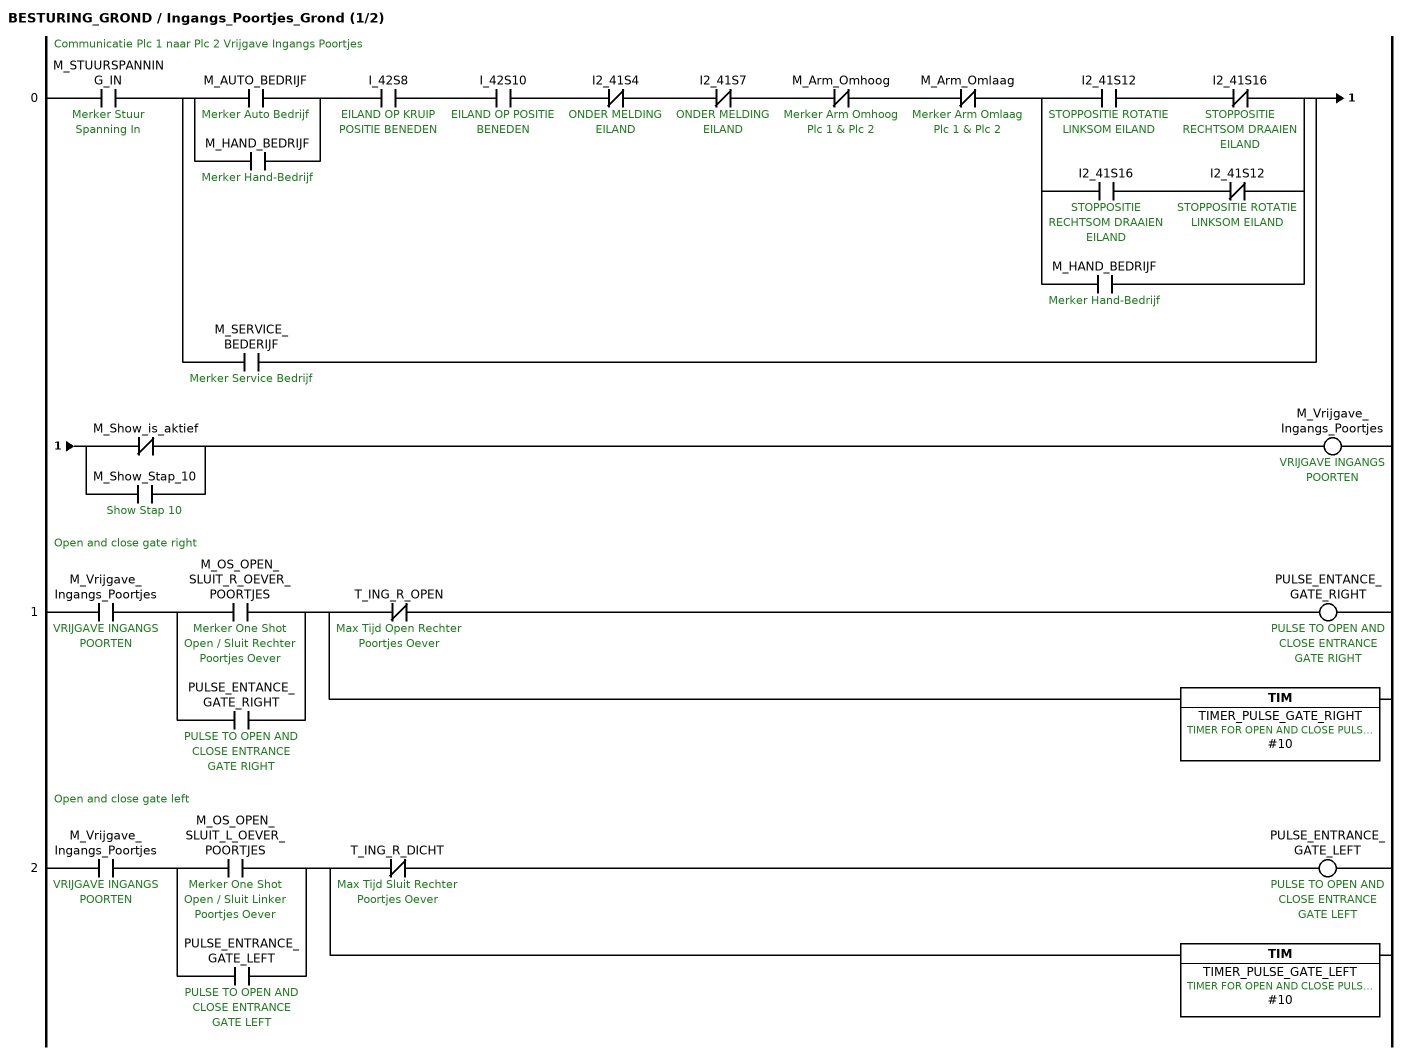
; [picture p349: BESTURING_GROND / Ingangs_Poortjes_Grond, rungs 0-2]
; rung 0: Communicatie Plc 1 naar Plc 2 Vrijgave Ingangs Poortjes
LD M_STUURSPANNING_IN  ; Merker Stuur Spanning In
LD M_AUTO_BEDRIJF  ; Merker Auto Bedrijf
OR M_HAND_BEDRIJF  ; Merker Hand-Bedrijf
AND I_42S8  ; EILAND OP KRUIP POSITIE BENEDEN
AND I_42S10  ; EILAND OP POSITIE BENEDEN
ANDNOT I2_41S4  ; ONDER MELDING EILAND
ANDNOT I2_41S7  ; ONDER MELDING EILAND
ANDNOT M_Arm_Omhoog  ; Merker Arm Omhoog Plc 1 & Plc 2
ANDNOT M_Arm_Omlaag  ; Merker Arm Omlaag Plc 1 & Plc 2
LD I2_41S12  ; STOPPOSITIE ROTATIE LINKSOM EILAND
ANDNOT I2_41S16  ; STOPPOSITIE RECHTSOM DRAAIEN EILAND
LD I2_41S16  ; STOPPOSITIE RECHTSOM DRAAIEN EILAND
ANDNOT I2_41S12  ; STOPPOSITIE ROTATIE LINKSOM EILAND
ORLD
OR M_HAND_BEDRIJF  ; Merker Hand-Bedrijf
ANDLD
OR M_SERVICE_BEDERIJF  ; Merker Service Bedrijf
ANDLD
LDNOT M_Show_is_aktief
OR M_Show_Stap_10  ; Show Stap 10
ANDLD
OUT M_Vrijgave_Ingangs_Poortjes  ; VRIJGAVE INGANGS POORTEN
; rung 1: Open and close gate right
LD M_Vrijgave_Ingangs_Poortjes  ; VRIJGAVE INGANGS POORTEN
LD M_OS_OPEN_SLUIT_R_OEVER_POORTJES  ; Merker One Shot Open / Sluit Rechter Poortjes Oever
OR PULSE_ENTANCE_GATE_RIGHT  ; PULSE TO OPEN AND CLOSE ENTRANCE GATE RIGHT
ANDLD
OUT TR0
ANDNOT T_ING_R_OPEN  ; Max Tijd Open Rechter Poortjes Oever
OUT PULSE_ENTANCE_GATE_RIGHT  ; PULSE TO OPEN AND CLOSE ENTRANCE GATE RIGHT
LD TR0
TIM TIMER_PULSE_GATE_RIGHT #10  ; TIMER FOR OPEN AND CLOSE PULSE ENTRANCE GATE RIGHT
; rung 2: Open and close gate left
LD M_Vrijgave_Ingangs_Poortjes  ; VRIJGAVE INGANGS POORTEN
LD M_OS_OPEN_SLUIT_L_OEVER_POORTJES  ; Merker One Shot Open / Sluit Linker Poortjes Oever
OR PULSE_ENTRANCE_GATE_LEFT  ; PULSE TO OPEN AND CLOSE ENTRANCE GATE LEFT
ANDLD
OUT TR0
ANDNOT T_ING_R_DICHT  ; Max Tijd Sluit Rechter Poortjes Oever
OUT PULSE_ENTRANCE_GATE_LEFT  ; PULSE TO OPEN AND CLOSE ENTRANCE GATE LEFT
LD TR0
TIM TIMER_PULSE_GATE_LEFT #10  ; TIMER FOR OPEN AND CLOSE PULSE ENTRANCE GATE LEFT

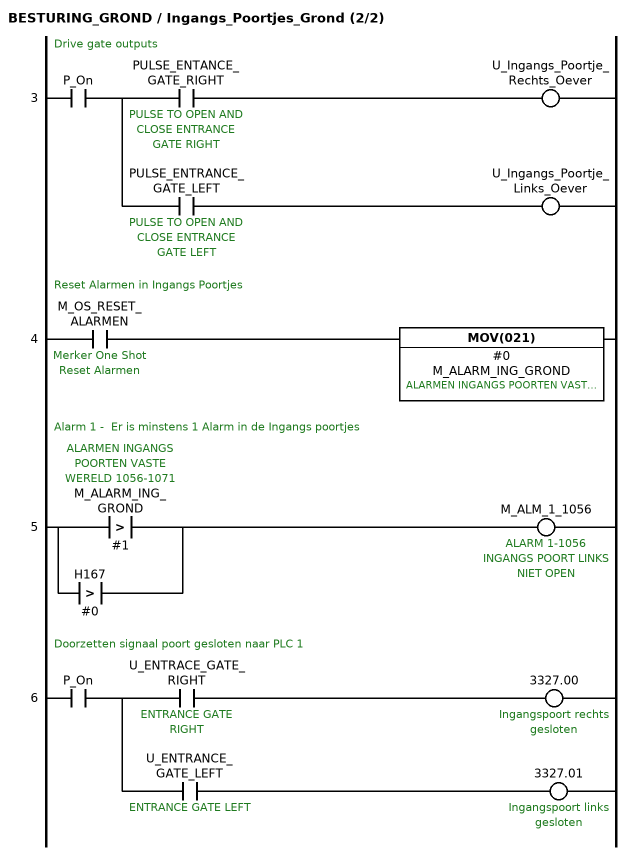
; rung 3: Drive gate outputs
LD P_On
OUT TR0
AND PULSE_ENTANCE_GATE_RIGHT  ; PULSE TO OPEN AND CLOSE ENTRANCE GATE RIGHT
OUT U_Ingangs_Poortje_Rechts_Oever
LD TR0
AND PULSE_ENTRANCE_GATE_LEFT  ; PULSE TO OPEN AND CLOSE ENTRANCE GATE LEFT
OUT U_Ingangs_Poortje_Links_Oever
; rung 4: Reset Alarmen in Ingangs Poortjes
LD M_OS_RESET_ALARMEN  ; Merker One Shot Reset Alarmen
MOV(021) #0 M_ALARM_ING_GROND  ; ALARMEN INGANGS POORTEN VASTE WERELD 1056-1071
; rung 5: Alarm 1 -  Er is minstens 1 Alarm in de Ingangs poortjes
LD>(320) M_ALARM_ING_GROND #1  ; ALARMEN INGANGS POORTEN VASTE WERELD 1056-1071
OR>(320) H167 #0
OUT M_ALM_1_1056  ; ALARM 1-1056 INGANGS POORT LINKS NIET OPEN
; rung 6: Doorzetten signaal poort gesloten naar PLC 1
LD P_On
OUT TR0
AND U_ENTRACE_GATE_RIGHT  ; ENTRANCE GATE RIGHT
OUT 3327.00  ; Ingangspoort rechts gesloten
LD TR0
AND U_ENTRANCE_GATE_LEFT  ; ENTRANCE GATE LEFT
OUT 3327.01  ; Ingangspoort links gesloten

### Section Uitgangs_poortjes_Grond

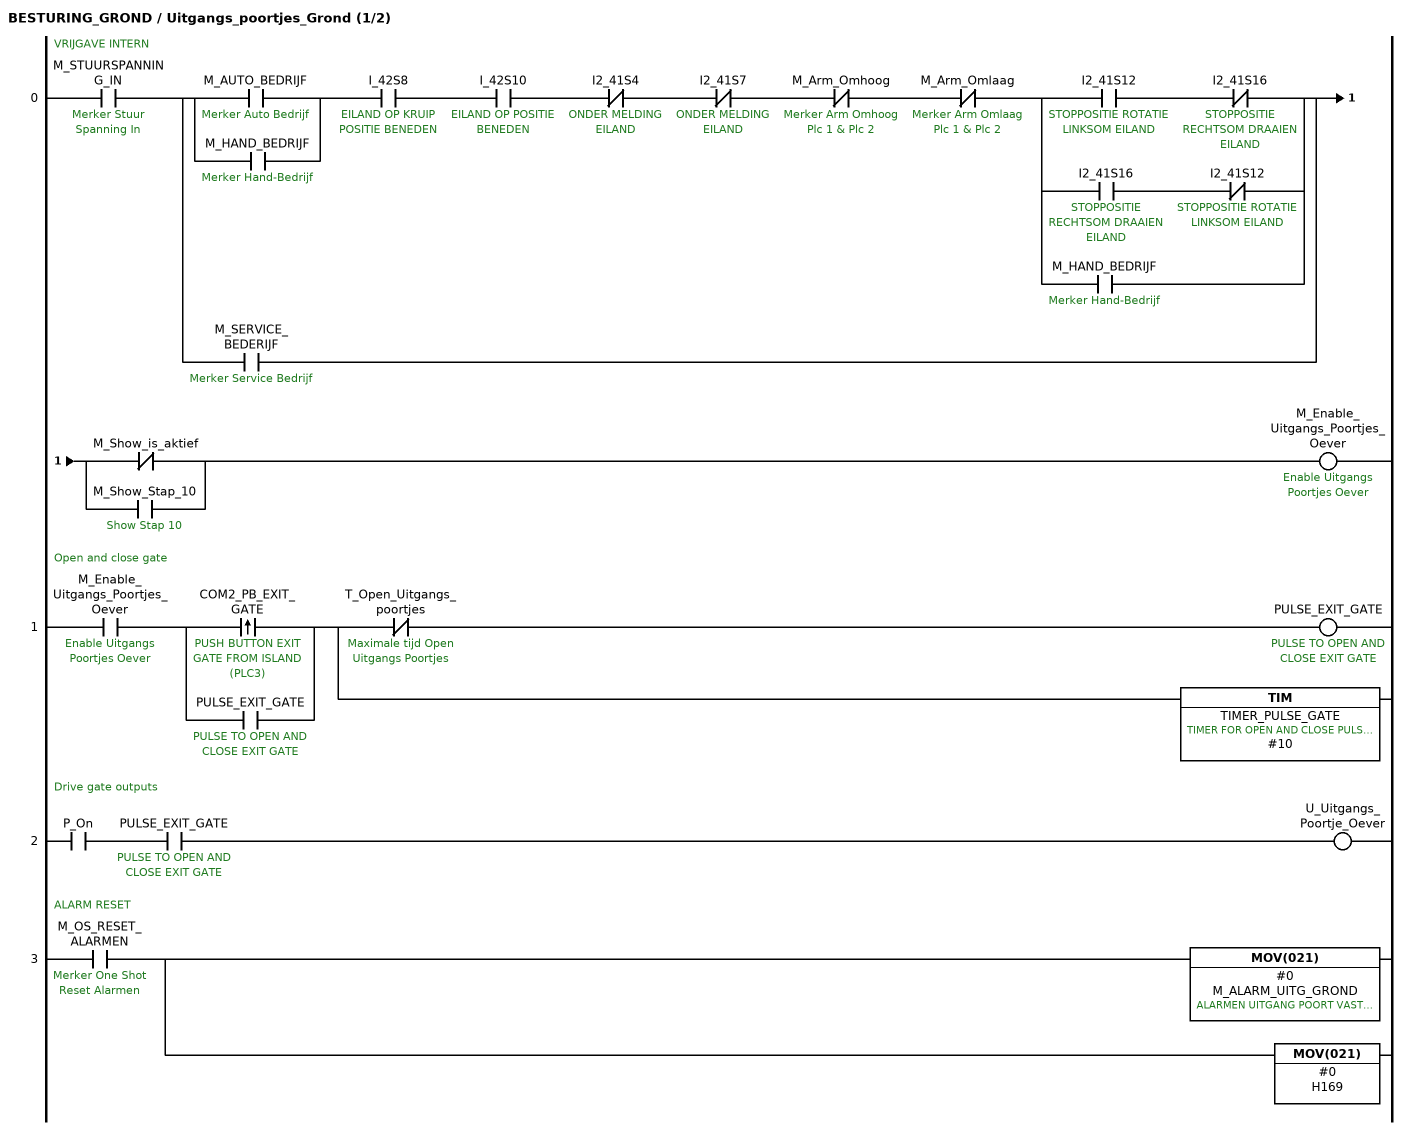
; rung 0: VRIJGAVE INTERN
LD M_STUURSPANNING_IN  ; Merker Stuur Spanning In
LD M_AUTO_BEDRIJF  ; Merker Auto Bedrijf
OR M_HAND_BEDRIJF  ; Merker Hand-Bedrijf
AND I_42S8  ; EILAND OP KRUIP POSITIE BENEDEN
AND I_42S10  ; EILAND OP POSITIE BENEDEN
ANDNOT I2_41S4  ; ONDER MELDING EILAND
ANDNOT I2_41S7  ; ONDER MELDING EILAND
ANDNOT M_Arm_Omhoog  ; Merker Arm Omhoog Plc 1 & Plc 2
ANDNOT M_Arm_Omlaag  ; Merker Arm Omlaag Plc 1 & Plc 2
LD I2_41S12  ; STOPPOSITIE ROTATIE LINKSOM EILAND
ANDNOT I2_41S16  ; STOPPOSITIE RECHTSOM DRAAIEN EILAND
LD I2_41S16  ; STOPPOSITIE RECHTSOM DRAAIEN EILAND
ANDNOT I2_41S12  ; STOPPOSITIE ROTATIE LINKSOM EILAND
ORLD
OR M_HAND_BEDRIJF  ; Merker Hand-Bedrijf
ANDLD
OR M_SERVICE_BEDERIJF  ; Merker Service Bedrijf
ANDLD
LDNOT M_Show_is_aktief
OR M_Show_Stap_10  ; Show Stap 10
ANDLD
OUT M_Enable_Uitgangs_Poortjes_Oever  ; Enable Uitgangs Poortjes Oever
; rung 1: Open and close gate
LD M_Enable_Uitgangs_Poortjes_Oever  ; Enable Uitgangs Poortjes Oever
@LD COM2_PB_EXIT_GATE  ; PUSH BUTTON EXIT GATE FROM ISLAND (PLC3)
OR PULSE_EXIT_GATE  ; PULSE TO OPEN AND CLOSE EXIT GATE
ANDLD
OUT TR0
ANDNOT T_Open_Uitgangs_poortjes  ; Maximale tijd Open Uitgangs Poortjes
OUT PULSE_EXIT_GATE  ; PULSE TO OPEN AND CLOSE EXIT GATE
LD TR0
TIM TIMER_PULSE_GATE #10  ; TIMER FOR OPEN AND CLOSE PULSE EXIT GATE
; rung 2: Drive gate outputs
LD P_On
AND PULSE_EXIT_GATE  ; PULSE TO OPEN AND CLOSE EXIT GATE
OUT U_Uitgangs_Poortje_Oever
; rung 3: ALARM RESET
LD M_OS_RESET_ALARMEN  ; Merker One Shot Reset Alarmen
MOV(021) #0 M_ALARM_UITG_GROND  ; ALARMEN UITGANG POORT VASTE WERELD 1088-1103
MOV(021) #0 H169

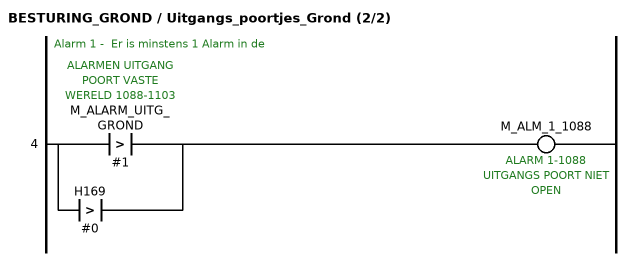
; rung 4: Alarm 1 -  Er is minstens 1 Alarm in de
LD>(320) M_ALARM_UITG_GROND #1  ; ALARMEN UITGANG POORT VASTE WERELD 1088-1103
OR>(320) H169 #0
OUT M_ALM_1_1088  ; ALARM 1-1088 UITGANGS POORT NIET OPEN

### Section Hydrauliek_Arm

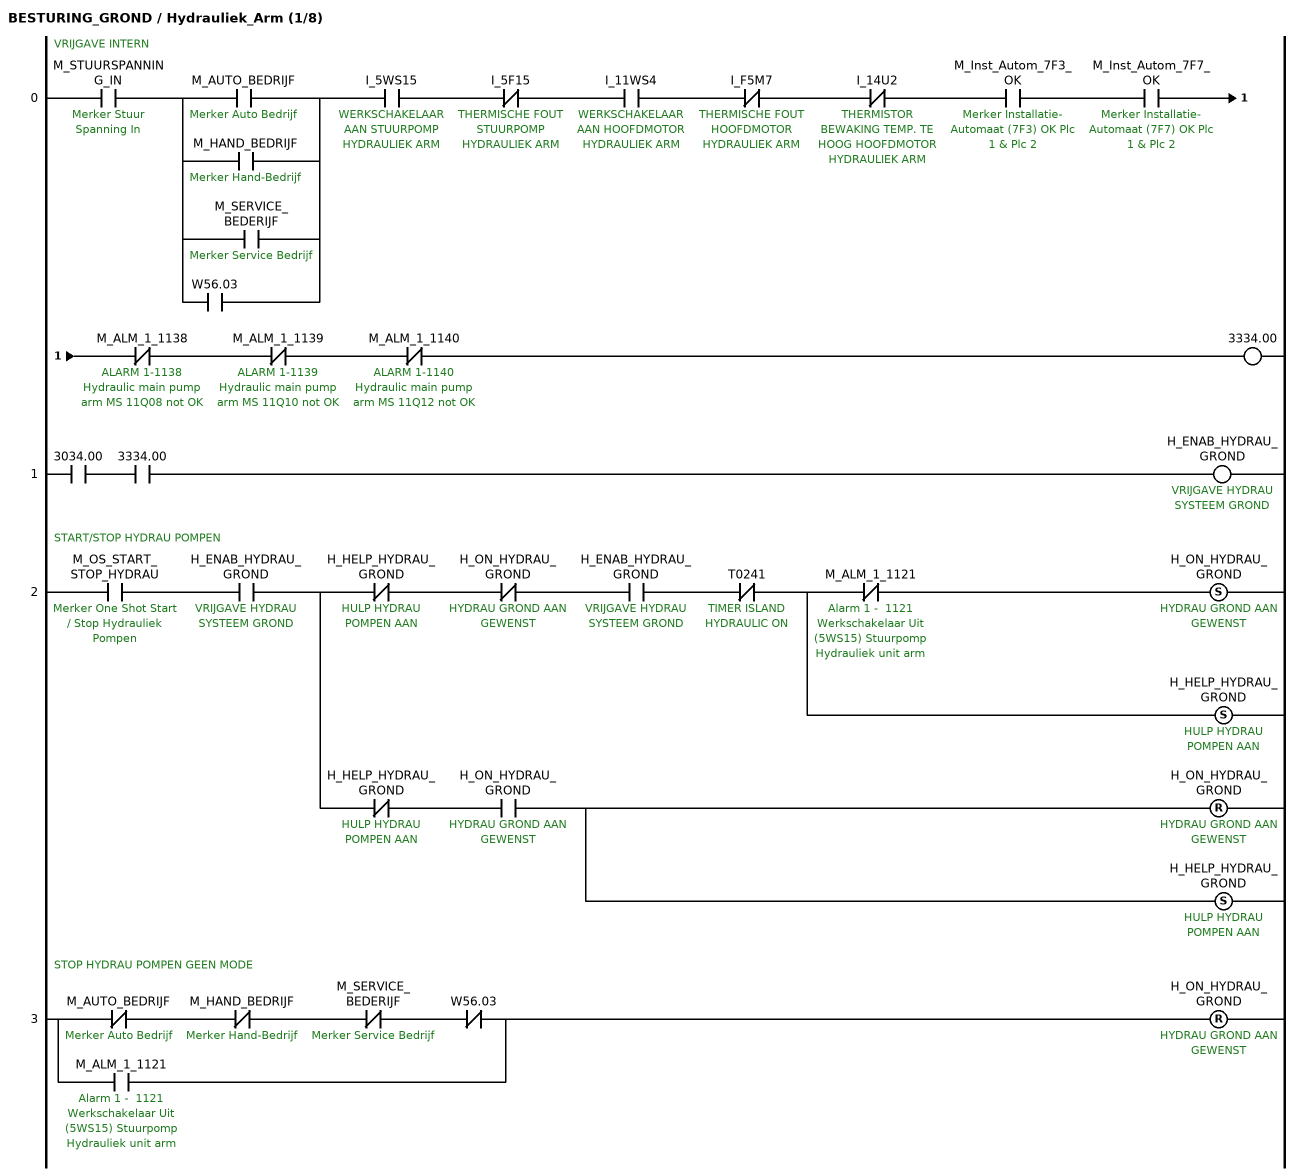
; rung 0: VRIJGAVE INTERN
LD M_STUURSPANNING_IN  ; Merker Stuur Spanning In
LD M_AUTO_BEDRIJF  ; Merker Auto Bedrijf
OR M_HAND_BEDRIJF  ; Merker Hand-Bedrijf
OR M_SERVICE_BEDERIJF  ; Merker Service Bedrijf
OR W56.03
ANDLD
AND I_5WS15  ; WERKSCHAKELAAR AAN STUURPOMP HYDRAULIEK ARM
ANDNOT I_5F15  ; THERMISCHE FOUT STUURPOMP HYDRAULIEK ARM
AND I_11WS4  ; WERKSCHAKELAAR AAN HOOFDMOTOR HYDRAULIEK ARM
ANDNOT I_F5M7  ; THERMISCHE FOUT HOOFDMOTOR HYDRAULIEK ARM
ANDNOT I_14U2  ; THERMISTOR BEWAKING TEMP. TE HOOG HOOFDMOTOR HYDRAULIEK ARM
AND M_Inst_Autom_7F3_OK  ; Merker Installatie-Automaat (7F3) OK Plc 1 & Plc 2
AND M_Inst_Autom_7F7_OK  ; Merker Installatie-Automaat (7F7) OK Plc 1 & Plc 2
ANDNOT M_ALM_1_1138  ; ALARM 1-1138 Hydraulic main pump arm MS 11Q08 not OK
ANDNOT M_ALM_1_1139  ; ALARM 1-1139 Hydraulic main pump arm MS 11Q10 not OK
ANDNOT M_ALM_1_1140  ; ALARM 1-1140 Hydraulic main pump arm MS 11Q12 not OK
OUT 3334.00
; rung 1
LD 3034.00
AND 3334.00
OUT H_ENAB_HYDRAU_GROND  ; VRIJGAVE HYDRAU SYSTEEM GROND
; rung 2: START/STOP HYDRAU POMPEN
LD M_OS_START_STOP_HYDRAU  ; Merker One Shot Start / Stop Hydrauliek Pompen
AND H_ENAB_HYDRAU_GROND  ; VRIJGAVE HYDRAU SYSTEEM GROND
OUT TR0
ANDNOT H_HELP_HYDRAU_GROND  ; HULP HYDRAU POMPEN AAN
ANDNOT H_ON_HYDRAU_GROND  ; HYDRAU GROND AAN GEWENST
AND H_ENAB_HYDRAU_GROND  ; VRIJGAVE HYDRAU SYSTEEM GROND
ANDNOT T0241  ; TIMER ISLAND HYDRAULIC ON
OUT TR1
ANDNOT M_ALM_1_1121  ; Alarm 1 -  1121 Werkschakelaar Uit (5WS15) Stuurpomp Hydrauliek unit arm
SET H_ON_HYDRAU_GROND  ; HYDRAU GROND AAN GEWENST
LD TR1
SET H_HELP_HYDRAU_GROND  ; HULP HYDRAU POMPEN AAN
LD TR0
ANDNOT H_HELP_HYDRAU_GROND  ; HULP HYDRAU POMPEN AAN
AND H_ON_HYDRAU_GROND  ; HYDRAU GROND AAN GEWENST
RSET H_ON_HYDRAU_GROND  ; HYDRAU GROND AAN GEWENST
SET H_HELP_HYDRAU_GROND  ; HULP HYDRAU POMPEN AAN
; rung 3: STOP HYDRAU POMPEN GEEN MODE
LDNOT M_AUTO_BEDRIJF  ; Merker Auto Bedrijf
ANDNOT M_HAND_BEDRIJF  ; Merker Hand-Bedrijf
ANDNOT M_SERVICE_BEDERIJF  ; Merker Service Bedrijf
ANDNOT W56.03
OR M_ALM_1_1121  ; Alarm 1 -  1121 Werkschakelaar Uit (5WS15) Stuurpomp Hydrauliek unit arm
RSET H_ON_HYDRAU_GROND  ; HYDRAU GROND AAN GEWENST

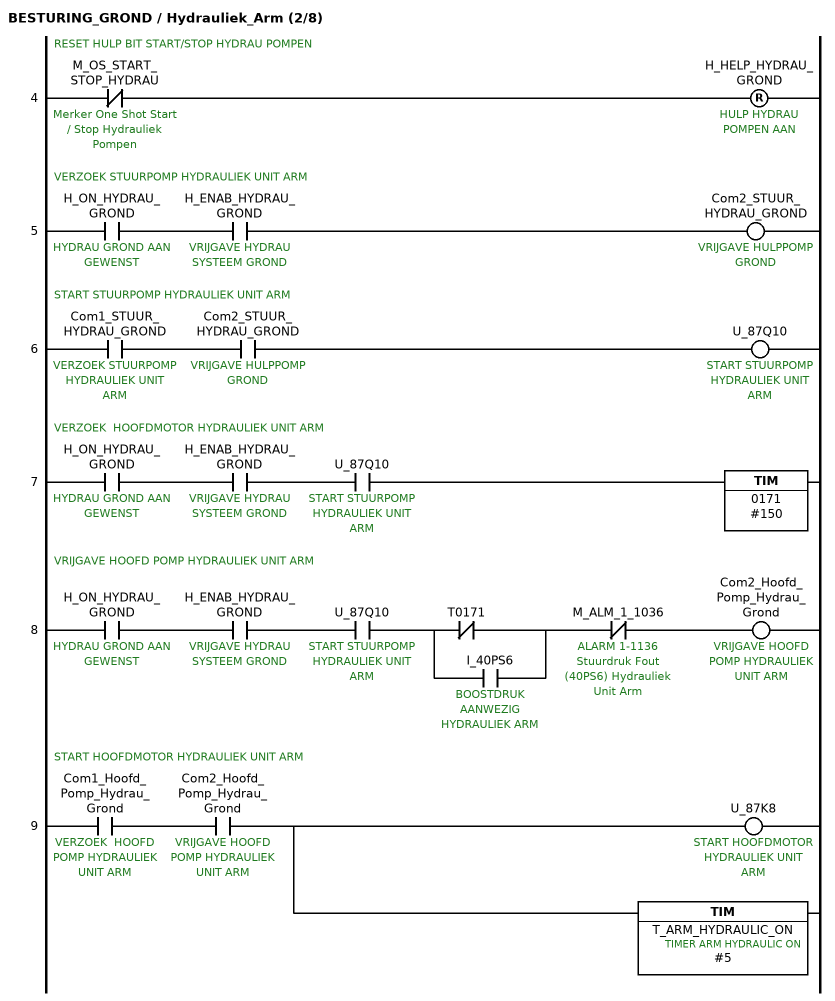
; rung 4: RESET HULP BIT START/STOP HYDRAU POMPEN
LDNOT M_OS_START_STOP_HYDRAU  ; Merker One Shot Start / Stop Hydrauliek Pompen
RSET H_HELP_HYDRAU_GROND  ; HULP HYDRAU POMPEN AAN
; rung 5: VERZOEK STUURPOMP HYDRAULIEK UNIT ARM
LD H_ON_HYDRAU_GROND  ; HYDRAU GROND AAN GEWENST
AND H_ENAB_HYDRAU_GROND  ; VRIJGAVE HYDRAU SYSTEEM GROND
OUT Com2_STUUR_HYDRAU_GROND  ; VRIJGAVE HULPPOMP GROND
; rung 6: START STUURPOMP HYDRAULIEK UNIT ARM
LD Com1_STUUR_HYDRAU_GROND  ; VERZOEK STUURPOMP HYDRAULIEK UNIT ARM
AND Com2_STUUR_HYDRAU_GROND  ; VRIJGAVE HULPPOMP GROND
OUT U_87Q10  ; START STUURPOMP HYDRAULIEK UNIT ARM
; rung 7: VERZOEK  HOOFDMOTOR HYDRAULIEK UNIT ARM
LD H_ON_HYDRAU_GROND  ; HYDRAU GROND AAN GEWENST
AND H_ENAB_HYDRAU_GROND  ; VRIJGAVE HYDRAU SYSTEEM GROND
AND U_87Q10  ; START STUURPOMP HYDRAULIEK UNIT ARM
TIM 0171 #150
; rung 8: VRIJGAVE HOOFD POMP HYDRAULIEK UNIT ARM
LD H_ON_HYDRAU_GROND  ; HYDRAU GROND AAN GEWENST
AND H_ENAB_HYDRAU_GROND  ; VRIJGAVE HYDRAU SYSTEEM GROND
AND U_87Q10  ; START STUURPOMP HYDRAULIEK UNIT ARM
LDNOT T0171
OR I_40PS6  ; BOOSTDRUK AANWEZIG HYDRAULIEK ARM
ANDLD
ANDNOT M_ALM_1_1036  ; ALARM 1-1136 Stuurdruk Fout (40PS6) Hydrauliek Unit Arm
OUT Com2_Hoofd_Pomp_Hydrau_Grond  ; VRIJGAVE HOOFD POMP HYDRAULIEK UNIT ARM
; rung 9: START HOOFDMOTOR HYDRAULIEK UNIT ARM
LD Com1_Hoofd_Pomp_Hydrau_Grond  ; VERZOEK  HOOFD POMP HYDRAULIEK UNIT ARM
AND Com2_Hoofd_Pomp_Hydrau_Grond  ; VRIJGAVE HOOFD POMP HYDRAULIEK UNIT ARM
OUT U_87K8  ; START HOOFDMOTOR HYDRAULIEK UNIT ARM
TIM T_ARM_HYDRAULIC_ON #5  ; TIMER ARM HYDRAULIC ON

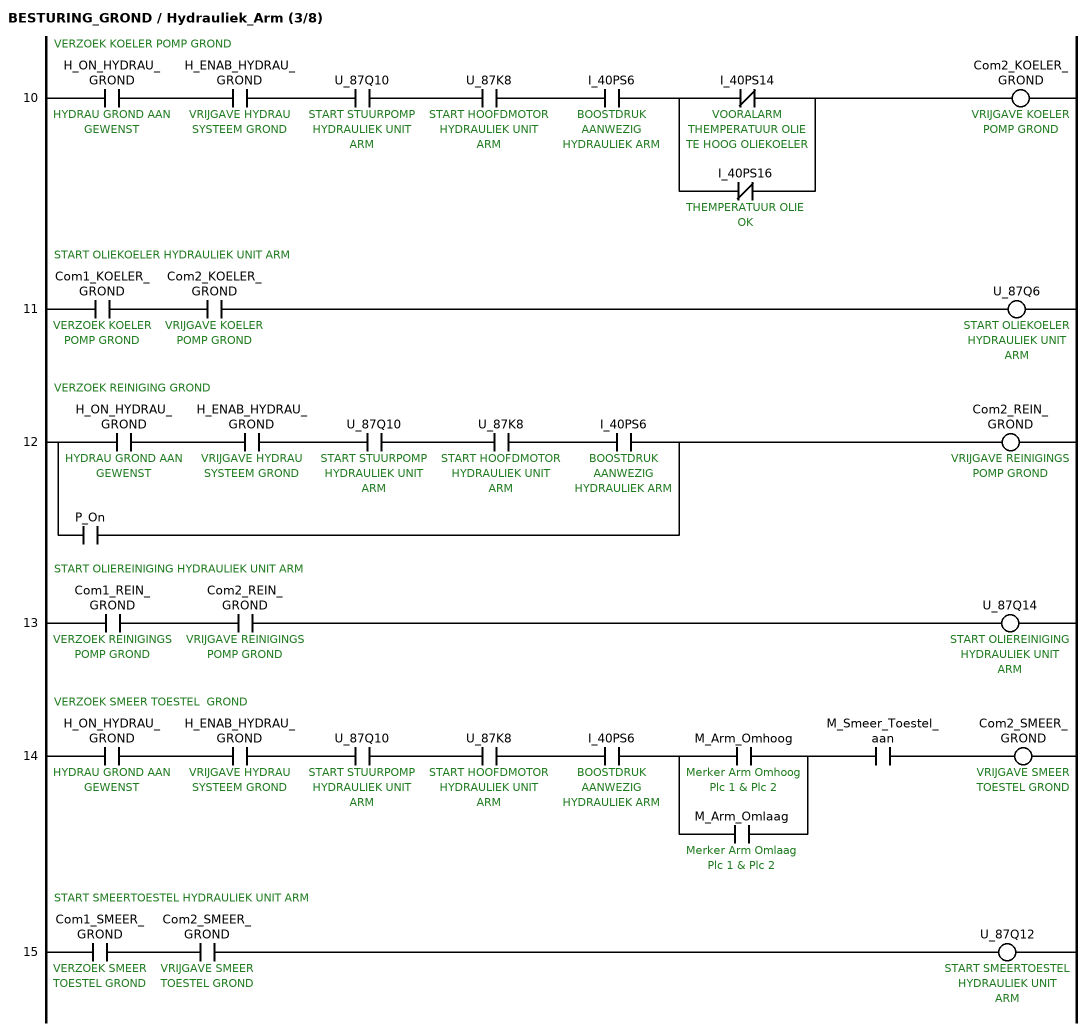
; rung 10: VERZOEK KOELER POMP GROND
LD H_ON_HYDRAU_GROND  ; HYDRAU GROND AAN GEWENST
AND H_ENAB_HYDRAU_GROND  ; VRIJGAVE HYDRAU SYSTEEM GROND
AND U_87Q10  ; START STUURPOMP HYDRAULIEK UNIT ARM
AND U_87K8  ; START HOOFDMOTOR HYDRAULIEK UNIT ARM
AND I_40PS6  ; BOOSTDRUK AANWEZIG HYDRAULIEK ARM
LDNOT I_40PS14  ; VOORALARM THEMPERATUUR OLIE TE HOOG OLIEKOELER
ORNOT I_40PS16  ; THEMPERATUUR OLIE OK
ANDLD
OUT Com2_KOELER_GROND  ; VRIJGAVE KOELER POMP GROND
; rung 11: START OLIEKOELER HYDRAULIEK UNIT ARM
LD Com1_KOELER_GROND  ; VERZOEK KOELER POMP GROND
AND Com2_KOELER_GROND  ; VRIJGAVE KOELER POMP GROND
OUT U_87Q6  ; START OLIEKOELER HYDRAULIEK UNIT ARM
; rung 12: VERZOEK REINIGING GROND
LD H_ON_HYDRAU_GROND  ; HYDRAU GROND AAN GEWENST
AND H_ENAB_HYDRAU_GROND  ; VRIJGAVE HYDRAU SYSTEEM GROND
AND U_87Q10  ; START STUURPOMP HYDRAULIEK UNIT ARM
AND U_87K8  ; START HOOFDMOTOR HYDRAULIEK UNIT ARM
AND I_40PS6  ; BOOSTDRUK AANWEZIG HYDRAULIEK ARM
OR P_On
OUT Com2_REIN_GROND  ; VRIJGAVE REINIGINGS POMP GROND
; rung 13: START OLIEREINIGING HYDRAULIEK UNIT ARM
LD Com1_REIN_GROND  ; VERZOEK REINIGINGS POMP GROND
AND Com2_REIN_GROND  ; VRIJGAVE REINIGINGS POMP GROND
OUT U_87Q14  ; START OLIEREINIGING HYDRAULIEK UNIT ARM
; rung 14: VERZOEK SMEER TOESTEL  GROND
LD H_ON_HYDRAU_GROND  ; HYDRAU GROND AAN GEWENST
AND H_ENAB_HYDRAU_GROND  ; VRIJGAVE HYDRAU SYSTEEM GROND
AND U_87Q10  ; START STUURPOMP HYDRAULIEK UNIT ARM
AND U_87K8  ; START HOOFDMOTOR HYDRAULIEK UNIT ARM
AND I_40PS6  ; BOOSTDRUK AANWEZIG HYDRAULIEK ARM
LD M_Arm_Omhoog  ; Merker Arm Omhoog Plc 1 & Plc 2
OR M_Arm_Omlaag  ; Merker Arm Omlaag Plc 1 & Plc 2
ANDLD
AND M_Smeer_Toestel_aan
OUT Com2_SMEER_GROND  ; VRIJGAVE SMEER TOESTEL GROND
; rung 15: START SMEERTOESTEL HYDRAULIEK UNIT ARM
LD Com1_SMEER_GROND  ; VERZOEK SMEER TOESTEL GROND
AND Com2_SMEER_GROND  ; VRIJGAVE SMEER TOESTEL GROND
OUT U_87Q12  ; START SMEERTOESTEL HYDRAULIEK UNIT ARM

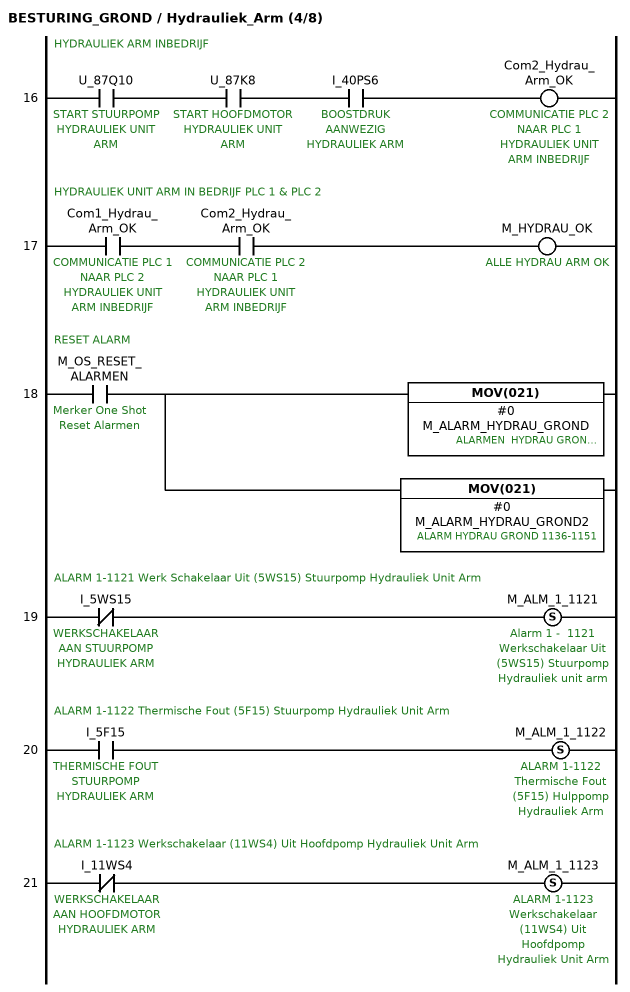
; rung 16: HYDRAULIEK ARM INBEDRIJF
LD U_87Q10  ; START STUURPOMP HYDRAULIEK UNIT ARM
AND U_87K8  ; START HOOFDMOTOR HYDRAULIEK UNIT ARM
AND I_40PS6  ; BOOSTDRUK AANWEZIG HYDRAULIEK ARM
OUT Com2_Hydrau_Arm_OK  ; COMMUNICATIE PLC 2 NAAR PLC 1 HYDRAULIEK UNIT ARM INBEDRIJF
; rung 17: HYDRAULIEK UNIT ARM IN BEDRIJF PLC 1 & PLC 2
LD Com1_Hydrau_Arm_OK  ; COMMUNICATIE PLC 1 NAAR PLC 2 HYDRAULIEK UNIT ARM INBEDRIJF
AND Com2_Hydrau_Arm_OK  ; COMMUNICATIE PLC 2 NAAR PLC 1 HYDRAULIEK UNIT ARM INBEDRIJF
OUT M_HYDRAU_OK  ; ALLE HYDRAU ARM OK
; rung 18: RESET ALARM
LD M_OS_RESET_ALARMEN  ; Merker One Shot Reset Alarmen
MOV(021) #0 M_ALARM_HYDRAU_GROND  ; ALARMEN  HYDRAU GROND 1120-1135
MOV(021) #0 M_ALARM_HYDRAU_GROND2  ; ALARM HYDRAU GROND 1136-1151
; rung 19: ALARM 1-1121 Werk Schakelaar Uit (5WS15) Stuurpomp Hydrauliek Unit Arm
LDNOT I_5WS15  ; WERKSCHAKELAAR AAN STUURPOMP HYDRAULIEK ARM
SET M_ALM_1_1121  ; Alarm 1 -  1121 Werkschakelaar Uit (5WS15) Stuurpomp Hydrauliek unit arm
; rung 20: ALARM 1-1122 Thermische Fout (5F15) Stuurpomp Hydrauliek Unit Arm
LD I_5F15  ; THERMISCHE FOUT STUURPOMP HYDRAULIEK ARM
SET M_ALM_1_1122  ; ALARM 1-1122 Thermische Fout (5F15) Hulppomp Hydrauliek Arm
; rung 21: ALARM 1-1123 Werkschakelaar (11WS4) Uit Hoofdpomp Hydrauliek Unit Arm
LDNOT I_11WS4  ; WERKSCHAKELAAR AAN HOOFDMOTOR HYDRAULIEK ARM
SET M_ALM_1_1123  ; ALARM 1-1123 Werkschakelaar (11WS4) Uit Hoofdpomp Hydrauliek Unit Arm

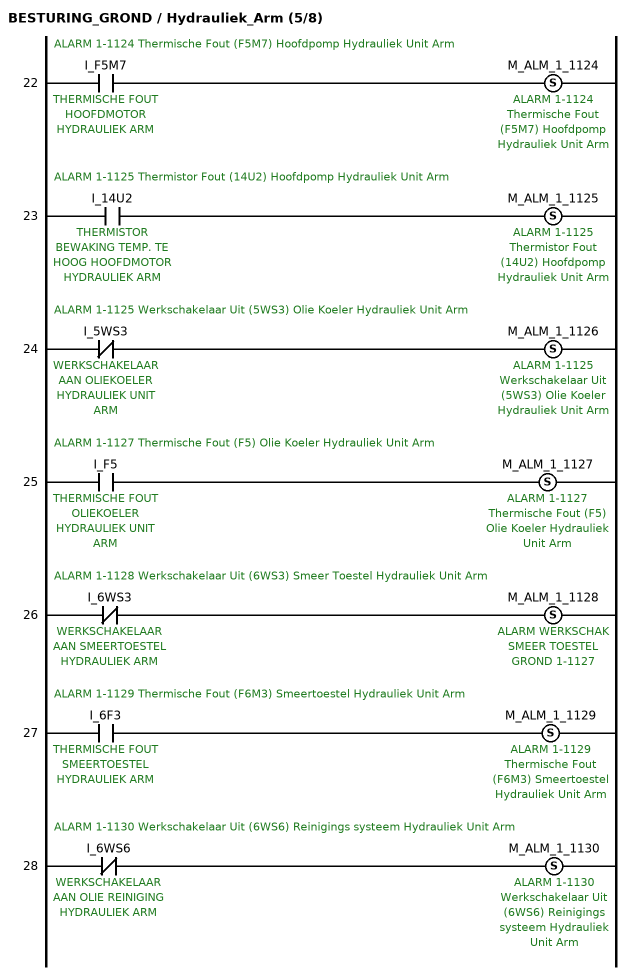
; rung 22: ALARM 1-1124 Thermische Fout (F5M7) Hoofdpomp Hydrauliek Unit Arm
LD I_F5M7  ; THERMISCHE FOUT HOOFDMOTOR HYDRAULIEK ARM
SET M_ALM_1_1124  ; ALARM 1-1124 Thermische Fout (F5M7) Hoofdpomp Hydrauliek Unit Arm
; rung 23: ALARM 1-1125 Thermistor Fout (14U2) Hoofdpomp Hydrauliek Unit Arm
LD I_14U2  ; THERMISTOR BEWAKING TEMP. TE HOOG HOOFDMOTOR HYDRAULIEK ARM
SET M_ALM_1_1125  ; ALARM 1-1125 Thermistor Fout (14U2) Hoofdpomp Hydrauliek Unit Arm
; rung 24: ALARM 1-1125 Werkschakelaar Uit (5WS3) Olie Koeler Hydrauliek Unit Arm
LDNOT I_5WS3  ; WERKSCHAKELAAR AAN OLIEKOELER HYDRAULIEK UNIT ARM
SET M_ALM_1_1126  ; ALARM 1-1125 Werkschakelaar Uit (5WS3) Olie Koeler Hydrauliek Unit Arm
; rung 25: ALARM 1-1127 Thermische Fout (F5) Olie Koeler Hydrauliek Unit Arm
LD I_F5  ; THERMISCHE FOUT OLIEKOELER HYDRAULIEK UNIT ARM
SET M_ALM_1_1127  ; ALARM 1-1127 Thermische Fout (F5) Olie Koeler Hydrauliek Unit Arm
; rung 26: ALARM 1-1128 Werkschakelaar Uit (6WS3) Smeer Toestel Hydrauliek Unit Arm
LDNOT I_6WS3  ; WERKSCHAKELAAR AAN SMEERTOESTEL HYDRAULIEK ARM
SET M_ALM_1_1128  ; ALARM WERKSCHAK SMEER TOESTEL GROND 1-1127
; rung 27: ALARM 1-1129 Thermische Fout (F6M3) Smeertoestel Hydrauliek Unit Arm
LD I_6F3  ; THERMISCHE FOUT SMEERTOESTEL HYDRAULIEK ARM
SET M_ALM_1_1129  ; ALARM 1-1129 Thermische Fout (F6M3) Smeertoestel Hydrauliek Unit Arm
; rung 28: ALARM 1-1130 Werkschakelaar Uit (6WS6) Reinigings systeem Hydrauliek Unit Arm
LDNOT I_6WS6  ; WERKSCHAKELAAR AAN OLIE REINIGING HYDRAULIEK ARM
SET M_ALM_1_1130  ; ALARM 1-1130 Werkschakelaar Uit (6WS6) Reinigings systeem Hydrauliek Unit Arm

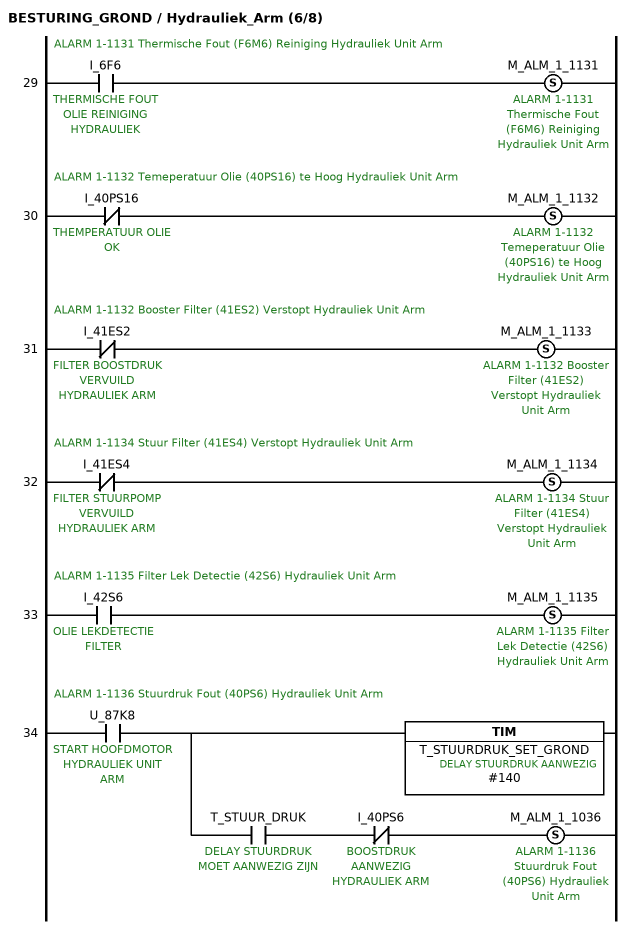
; rung 29: ALARM 1-1131 Thermische Fout (F6M6) Reiniging Hydrauliek Unit Arm
LD I_6F6  ; THERMISCHE FOUT OLIE REINIGING HYDRAULIEK
SET M_ALM_1_1131  ; ALARM 1-1131 Thermische Fout (F6M6) Reiniging Hydrauliek Unit Arm
; rung 30: ALARM 1-1132 Temeperatuur Olie (40PS16) te Hoog Hydrauliek Unit Arm
LDNOT I_40PS16  ; THEMPERATUUR OLIE OK
SET M_ALM_1_1132  ; ALARM 1-1132 Temeperatuur Olie (40PS16) te Hoog Hydrauliek Unit Arm
; rung 31: ALARM 1-1132 Booster Filter (41ES2) Verstopt Hydrauliek Unit Arm
LDNOT I_41ES2  ; FILTER BOOSTDRUK VERVUILD HYDRAULIEK ARM
SET M_ALM_1_1133  ; ALARM 1-1132 Booster Filter (41ES2) Verstopt Hydrauliek Unit Arm
; rung 32: ALARM 1-1134 Stuur Filter (41ES4) Verstopt Hydrauliek Unit Arm
LDNOT I_41ES4  ; FILTER STUURPOMP VERVUILD HYDRAULIEK ARM
SET M_ALM_1_1134  ; ALARM 1-1134 Stuur Filter (41ES4) Verstopt Hydrauliek Unit Arm
; rung 33: ALARM 1-1135 Filter Lek Detectie (42S6) Hydrauliek Unit Arm
LD I_42S6  ; OLIE LEKDETECTIE FILTER
SET M_ALM_1_1135  ; ALARM 1-1135 Filter Lek Detectie (42S6) Hydrauliek Unit Arm
; rung 34: ALARM 1-1136 Stuurdruk Fout (40PS6) Hydrauliek Unit Arm
LD U_87K8  ; START HOOFDMOTOR HYDRAULIEK UNIT ARM
TIM T_STUURDRUK_SET_GROND #140  ; DELAY STUURDRUK AANWEZIG
AND T_STUUR_DRUK  ; DELAY STUURDRUK MOET AANWEZIG ZIJN
ANDNOT I_40PS6  ; BOOSTDRUK AANWEZIG HYDRAULIEK ARM
SET M_ALM_1_1036  ; ALARM 1-1136 Stuurdruk Fout (40PS6) Hydrauliek Unit Arm

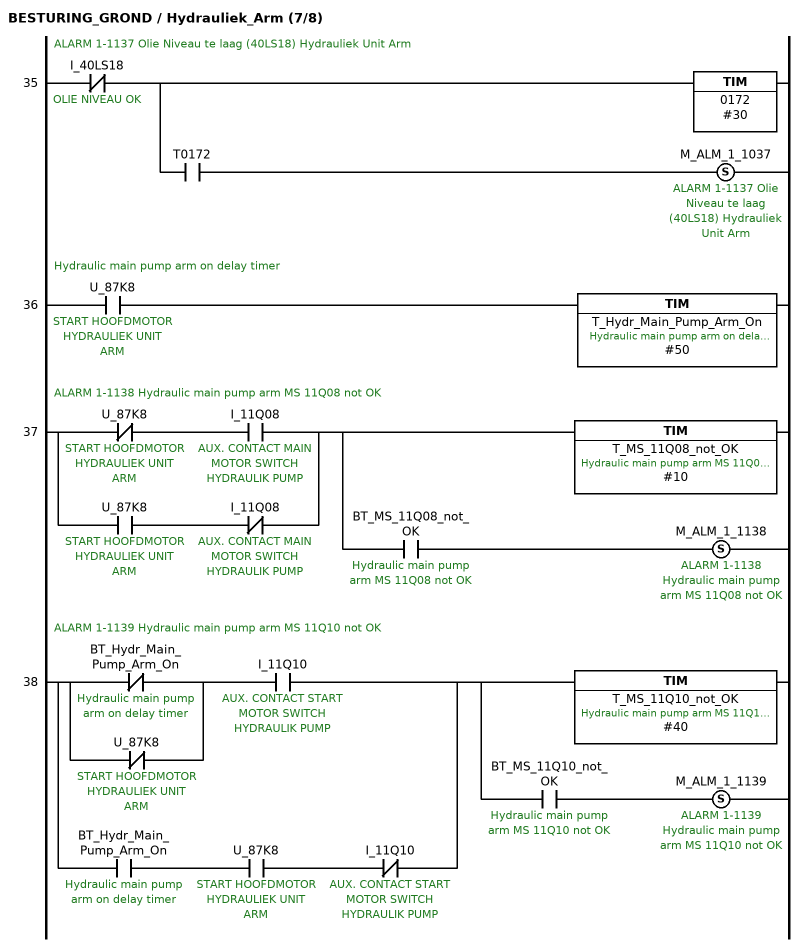
; rung 35: ALARM 1-1137 Olie Niveau te laag (40LS18) Hydrauliek Unit Arm
LDNOT I_40LS18  ; OLIE NIVEAU OK
TIM 0172 #30
AND T0172
SET M_ALM_1_1037  ; ALARM 1-1137 Olie Niveau te laag (40LS18) Hydrauliek Unit Arm
; rung 36: Hydraulic main pump arm on delay timer
LD U_87K8  ; START HOOFDMOTOR HYDRAULIEK UNIT ARM
TIM T_Hydr_Main_Pump_Arm_On #50  ; Hydraulic main pump arm on delay timer
; rung 37: ALARM 1-1138 Hydraulic main pump arm MS 11Q08 not OK
LDNOT U_87K8  ; START HOOFDMOTOR HYDRAULIEK UNIT ARM
AND I_11Q08  ; AUX. CONTACT MAIN MOTOR SWITCH HYDRAULIK PUMP
LD U_87K8  ; START HOOFDMOTOR HYDRAULIEK UNIT ARM
ANDNOT I_11Q08  ; AUX. CONTACT MAIN MOTOR SWITCH HYDRAULIK PUMP
ORLD
TIM T_MS_11Q08_not_OK #10  ; Hydraulic main pump arm MS 11Q08 not OK
AND BT_MS_11Q08_not_OK  ; Hydraulic main pump arm MS 11Q08 not OK
SET M_ALM_1_1138  ; ALARM 1-1138 Hydraulic main pump arm MS 11Q08 not OK
; rung 38: ALARM 1-1139 Hydraulic main pump arm MS 11Q10 not OK
LDNOT BT_Hydr_Main_Pump_Arm_On  ; Hydraulic main pump arm on delay timer
ORNOT U_87K8  ; START HOOFDMOTOR HYDRAULIEK UNIT ARM
AND I_11Q10  ; AUX. CONTACT START MOTOR SWITCH HYDRAULIK PUMP
LD BT_Hydr_Main_Pump_Arm_On  ; Hydraulic main pump arm on delay timer
AND U_87K8  ; START HOOFDMOTOR HYDRAULIEK UNIT ARM
ANDNOT I_11Q10  ; AUX. CONTACT START MOTOR SWITCH HYDRAULIK PUMP
ORLD
TIM T_MS_11Q10_not_OK #40  ; Hydraulic main pump arm MS 11Q10 not OK
AND BT_MS_11Q10_not_OK  ; Hydraulic main pump arm MS 11Q10 not OK
SET M_ALM_1_1139  ; ALARM 1-1139 Hydraulic main pump arm MS 11Q10 not OK

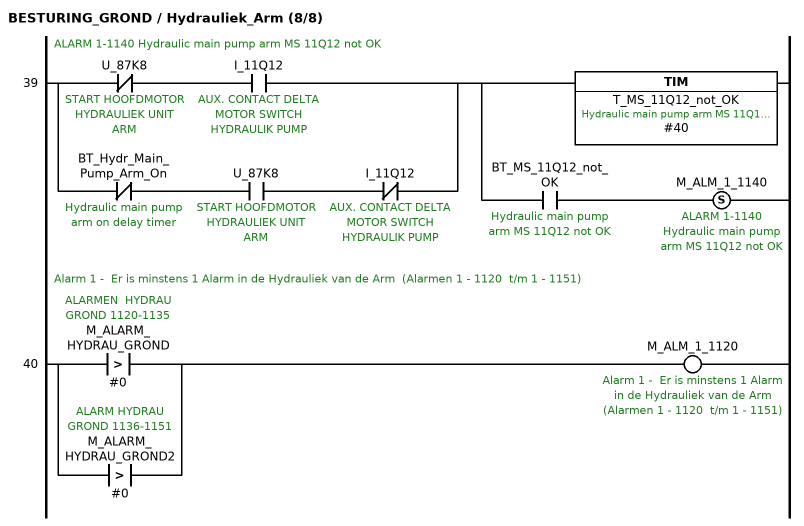
; rung 39: ALARM 1-1140 Hydraulic main pump arm MS 11Q12 not OK
LDNOT U_87K8  ; START HOOFDMOTOR HYDRAULIEK UNIT ARM
AND I_11Q12  ; AUX. CONTACT DELTA MOTOR SWITCH HYDRAULIK PUMP
LDNOT BT_Hydr_Main_Pump_Arm_On  ; Hydraulic main pump arm on delay timer
AND U_87K8  ; START HOOFDMOTOR HYDRAULIEK UNIT ARM
ANDNOT I_11Q12  ; AUX. CONTACT DELTA MOTOR SWITCH HYDRAULIK PUMP
ORLD
TIM T_MS_11Q12_not_OK #40  ; Hydraulic main pump arm MS 11Q12 not OK
AND BT_MS_11Q12_not_OK  ; Hydraulic main pump arm MS 11Q12 not OK
SET M_ALM_1_1140  ; ALARM 1-1140 Hydraulic main pump arm MS 11Q12 not OK
; rung 40: Alarm 1 -  Er is minstens 1 Alarm in de Hydrauliek van de Arm  (Alarmen 1 - 1120  t/m 1 - 1151)
LD>(320) M_ALARM_HYDRAU_GROND #0  ; ALARMEN  HYDRAU GROND 1120-1135
OR>(320) M_ALARM_HYDRAU_GROND2 #0  ; ALARM HYDRAU GROND 1136-1151
OUT M_ALM_1_1120  ; Alarm 1 -  Er is minstens 1 Alarm in de Hydrauliek van de Arm  (Alarmen 1 - 1120  t/m 1 - 1151)

### Section Data_Arm

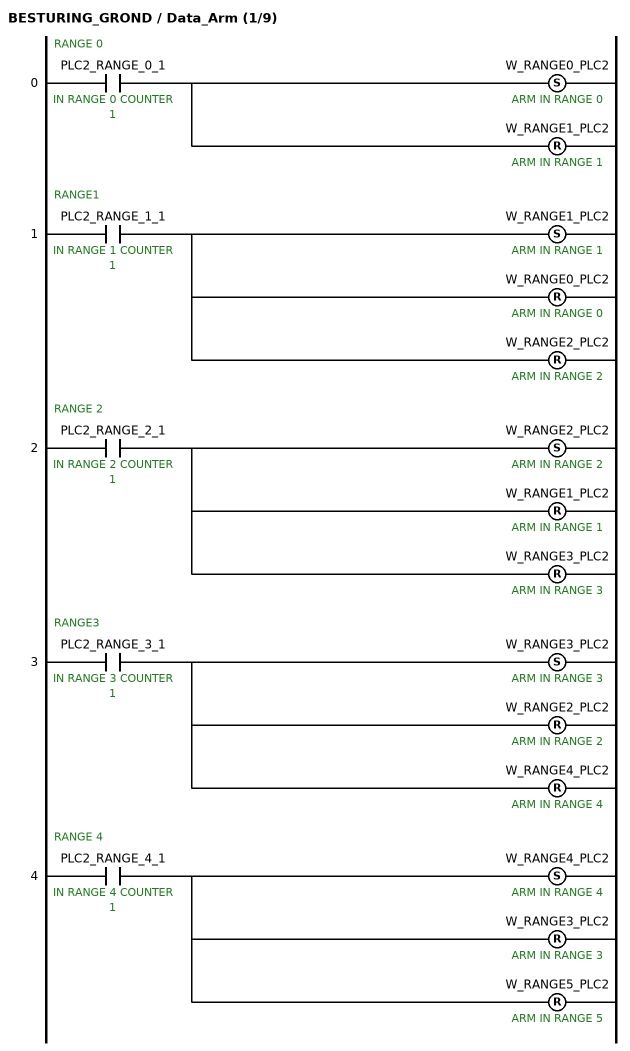
; rung 0: RANGE 0
LD PLC2_RANGE_0_1  ; IN RANGE 0 COUNTER 1
SET W_RANGE0_PLC2  ; ARM IN RANGE 0
RSET W_RANGE1_PLC2  ; ARM IN RANGE 1
; rung 1: RANGE1
LD PLC2_RANGE_1_1  ; IN RANGE 1 COUNTER 1
SET W_RANGE1_PLC2  ; ARM IN RANGE 1
RSET W_RANGE0_PLC2  ; ARM IN RANGE 0
RSET W_RANGE2_PLC2  ; ARM IN RANGE 2
; rung 2: RANGE 2
LD PLC2_RANGE_2_1  ; IN RANGE 2 COUNTER 1
SET W_RANGE2_PLC2  ; ARM IN RANGE 2
RSET W_RANGE1_PLC2  ; ARM IN RANGE 1
RSET W_RANGE3_PLC2  ; ARM IN RANGE 3
; rung 3: RANGE3
LD PLC2_RANGE_3_1  ; IN RANGE 3 COUNTER 1
SET W_RANGE3_PLC2  ; ARM IN RANGE 3
RSET W_RANGE2_PLC2  ; ARM IN RANGE 2
RSET W_RANGE4_PLC2  ; ARM IN RANGE 4
; rung 4: RANGE 4
LD PLC2_RANGE_4_1  ; IN RANGE 4 COUNTER 1
SET W_RANGE4_PLC2  ; ARM IN RANGE 4
RSET W_RANGE3_PLC2  ; ARM IN RANGE 3
RSET W_RANGE5_PLC2  ; ARM IN RANGE 5

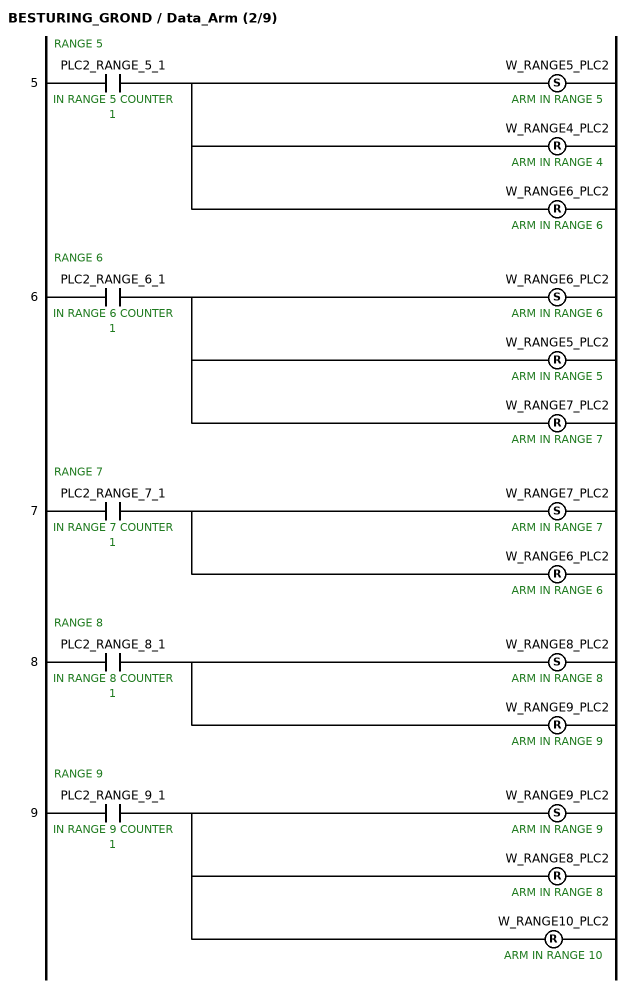
; rung 5: RANGE 5
LD PLC2_RANGE_5_1  ; IN RANGE 5 COUNTER 1
SET W_RANGE5_PLC2  ; ARM IN RANGE 5
RSET W_RANGE4_PLC2  ; ARM IN RANGE 4
RSET W_RANGE6_PLC2  ; ARM IN RANGE 6
; rung 6: RANGE 6
LD PLC2_RANGE_6_1  ; IN RANGE 6 COUNTER 1
SET W_RANGE6_PLC2  ; ARM IN RANGE 6
RSET W_RANGE5_PLC2  ; ARM IN RANGE 5
RSET W_RANGE7_PLC2  ; ARM IN RANGE 7
; rung 7: RANGE 7
LD PLC2_RANGE_7_1  ; IN RANGE 7 COUNTER 1
SET W_RANGE7_PLC2  ; ARM IN RANGE 7
RSET W_RANGE6_PLC2  ; ARM IN RANGE 6
; rung 8: RANGE 8
LD PLC2_RANGE_8_1  ; IN RANGE 8 COUNTER 1
SET W_RANGE8_PLC2  ; ARM IN RANGE 8
RSET W_RANGE9_PLC2  ; ARM IN RANGE 9
; rung 9: RANGE 9
LD PLC2_RANGE_9_1  ; IN RANGE 9 COUNTER 1
SET W_RANGE9_PLC2  ; ARM IN RANGE 9
RSET W_RANGE8_PLC2  ; ARM IN RANGE 8
RSET W_RANGE10_PLC2  ; ARM IN RANGE 10

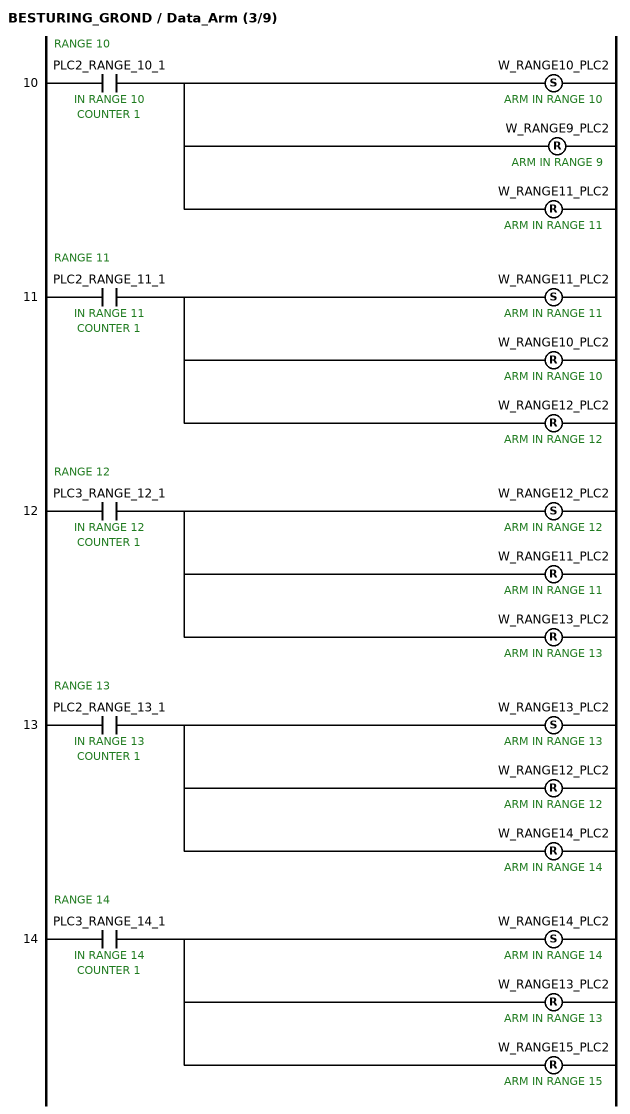
; rung 10: RANGE 10
LD PLC2_RANGE_10_1  ; IN RANGE 10 COUNTER 1
SET W_RANGE10_PLC2  ; ARM IN RANGE 10
RSET W_RANGE9_PLC2  ; ARM IN RANGE 9
RSET W_RANGE11_PLC2  ; ARM IN RANGE 11
; rung 11: RANGE 11
LD PLC2_RANGE_11_1  ; IN RANGE 11 COUNTER 1
SET W_RANGE11_PLC2  ; ARM IN RANGE 11
RSET W_RANGE10_PLC2  ; ARM IN RANGE 10
RSET W_RANGE12_PLC2  ; ARM IN RANGE 12
; rung 12: RANGE 12
LD PLC3_RANGE_12_1  ; IN RANGE 12 COUNTER 1
SET W_RANGE12_PLC2  ; ARM IN RANGE 12
RSET W_RANGE11_PLC2  ; ARM IN RANGE 11
RSET W_RANGE13_PLC2  ; ARM IN RANGE 13
; rung 13: RANGE 13
LD PLC2_RANGE_13_1  ; IN RANGE 13 COUNTER 1
SET W_RANGE13_PLC2  ; ARM IN RANGE 13
RSET W_RANGE12_PLC2  ; ARM IN RANGE 12
RSET W_RANGE14_PLC2  ; ARM IN RANGE 14
; rung 14: RANGE 14
LD PLC3_RANGE_14_1  ; IN RANGE 14 COUNTER 1
SET W_RANGE14_PLC2  ; ARM IN RANGE 14
RSET W_RANGE13_PLC2  ; ARM IN RANGE 13
RSET W_RANGE15_PLC2  ; ARM IN RANGE 15

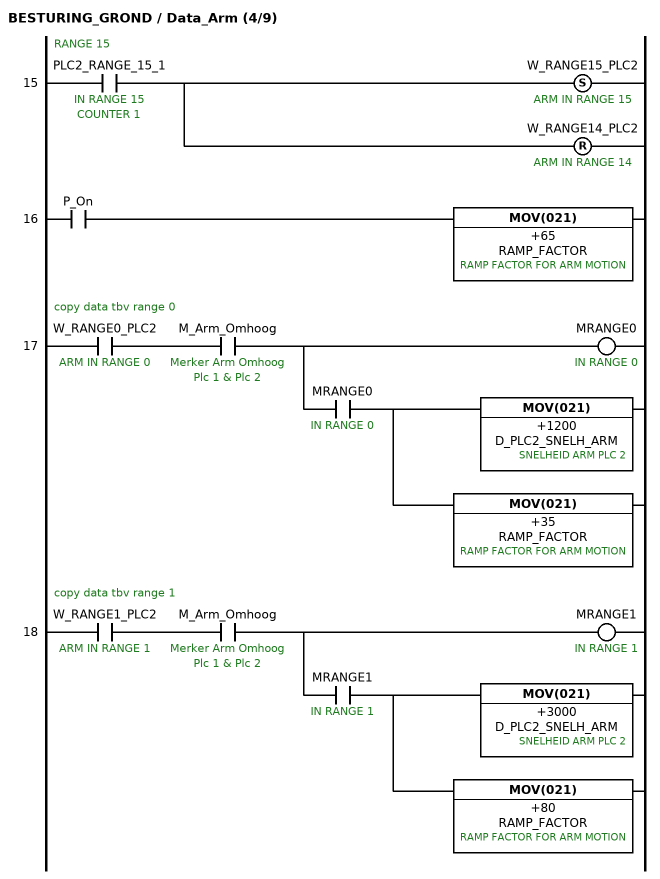
; rung 15: RANGE 15
LD PLC2_RANGE_15_1  ; IN RANGE 15 COUNTER 1
SET W_RANGE15_PLC2  ; ARM IN RANGE 15
RSET W_RANGE14_PLC2  ; ARM IN RANGE 14
; rung 16
LD P_On
MOV(021) +65 RAMP_FACTOR  ; RAMP FACTOR FOR ARM MOTION
; rung 17: copy data tbv range 0
LD W_RANGE0_PLC2  ; ARM IN RANGE 0
AND M_Arm_Omhoog  ; Merker Arm Omhoog Plc 1 & Plc 2
OUT MRANGE0  ; IN RANGE 0
AND MRANGE0  ; IN RANGE 0
MOV(021) +1200 D_PLC2_SNELH_ARM  ; SNELHEID ARM PLC 2
MOV(021) +35 RAMP_FACTOR  ; RAMP FACTOR FOR ARM MOTION
; rung 18: copy data tbv range 1
LD W_RANGE1_PLC2  ; ARM IN RANGE 1
AND M_Arm_Omhoog  ; Merker Arm Omhoog Plc 1 & Plc 2
OUT MRANGE1  ; IN RANGE 1
AND MRANGE1  ; IN RANGE 1
MOV(021) +3000 D_PLC2_SNELH_ARM  ; SNELHEID ARM PLC 2
MOV(021) +80 RAMP_FACTOR  ; RAMP FACTOR FOR ARM MOTION

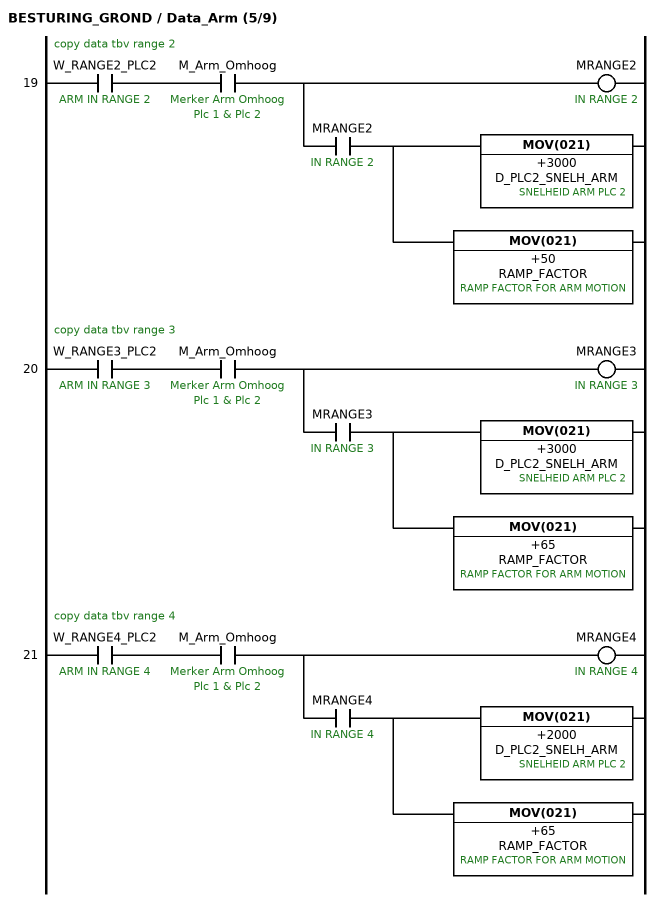
; rung 19: copy data tbv range 2
LD W_RANGE2_PLC2  ; ARM IN RANGE 2
AND M_Arm_Omhoog  ; Merker Arm Omhoog Plc 1 & Plc 2
OUT MRANGE2  ; IN RANGE 2
AND MRANGE2  ; IN RANGE 2
MOV(021) +3000 D_PLC2_SNELH_ARM  ; SNELHEID ARM PLC 2
MOV(021) +50 RAMP_FACTOR  ; RAMP FACTOR FOR ARM MOTION
; rung 20: copy data tbv range 3
LD W_RANGE3_PLC2  ; ARM IN RANGE 3
AND M_Arm_Omhoog  ; Merker Arm Omhoog Plc 1 & Plc 2
OUT MRANGE3  ; IN RANGE 3
AND MRANGE3  ; IN RANGE 3
MOV(021) +3000 D_PLC2_SNELH_ARM  ; SNELHEID ARM PLC 2
MOV(021) +65 RAMP_FACTOR  ; RAMP FACTOR FOR ARM MOTION
; rung 21: copy data tbv range 4
LD W_RANGE4_PLC2  ; ARM IN RANGE 4
AND M_Arm_Omhoog  ; Merker Arm Omhoog Plc 1 & Plc 2
OUT MRANGE4  ; IN RANGE 4
AND MRANGE4  ; IN RANGE 4
MOV(021) +2000 D_PLC2_SNELH_ARM  ; SNELHEID ARM PLC 2
MOV(021) +65 RAMP_FACTOR  ; RAMP FACTOR FOR ARM MOTION

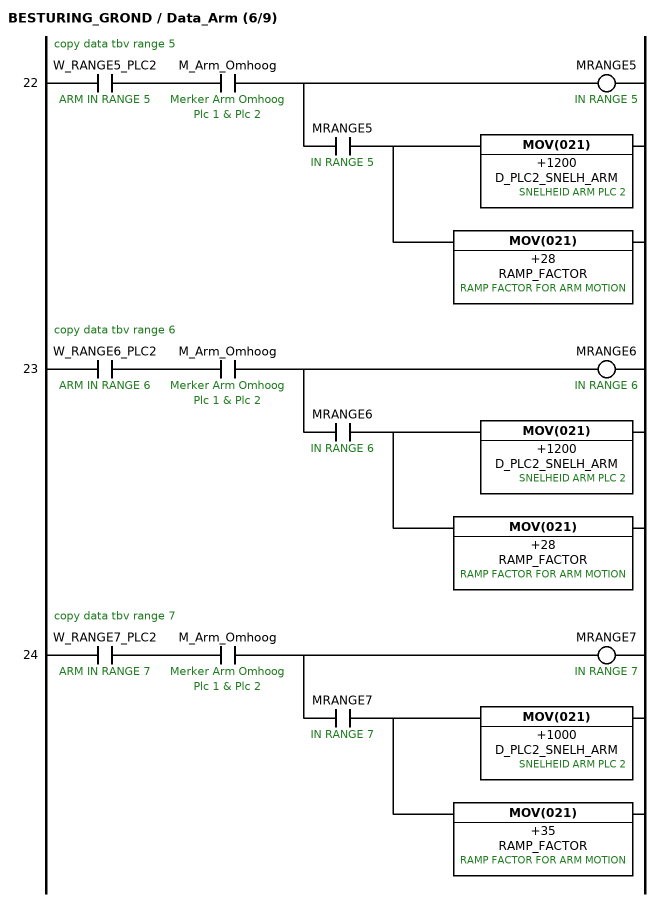
; rung 22: copy data tbv range 5
LD W_RANGE5_PLC2  ; ARM IN RANGE 5
AND M_Arm_Omhoog  ; Merker Arm Omhoog Plc 1 & Plc 2
OUT MRANGE5  ; IN RANGE 5
AND MRANGE5  ; IN RANGE 5
MOV(021) +1200 D_PLC2_SNELH_ARM  ; SNELHEID ARM PLC 2
MOV(021) +28 RAMP_FACTOR  ; RAMP FACTOR FOR ARM MOTION
; rung 23: copy data tbv range 6
LD W_RANGE6_PLC2  ; ARM IN RANGE 6
AND M_Arm_Omhoog  ; Merker Arm Omhoog Plc 1 & Plc 2
OUT MRANGE6  ; IN RANGE 6
AND MRANGE6  ; IN RANGE 6
MOV(021) +1200 D_PLC2_SNELH_ARM  ; SNELHEID ARM PLC 2
MOV(021) +28 RAMP_FACTOR  ; RAMP FACTOR FOR ARM MOTION
; rung 24: copy data tbv range 7
LD W_RANGE7_PLC2  ; ARM IN RANGE 7
AND M_Arm_Omhoog  ; Merker Arm Omhoog Plc 1 & Plc 2
OUT MRANGE7  ; IN RANGE 7
AND MRANGE7  ; IN RANGE 7
MOV(021) +1000 D_PLC2_SNELH_ARM  ; SNELHEID ARM PLC 2
MOV(021) +35 RAMP_FACTOR  ; RAMP FACTOR FOR ARM MOTION

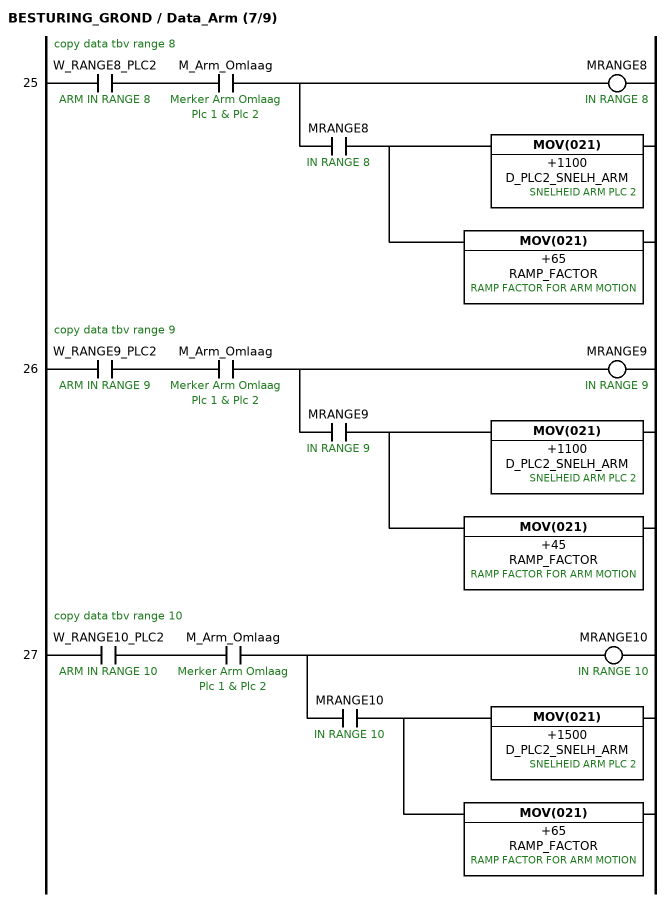
; rung 25: copy data tbv range 8
LD W_RANGE8_PLC2  ; ARM IN RANGE 8
AND M_Arm_Omlaag  ; Merker Arm Omlaag Plc 1 & Plc 2
OUT MRANGE8  ; IN RANGE 8
AND MRANGE8  ; IN RANGE 8
MOV(021) +1100 D_PLC2_SNELH_ARM  ; SNELHEID ARM PLC 2
MOV(021) +65 RAMP_FACTOR  ; RAMP FACTOR FOR ARM MOTION
; rung 26: copy data tbv range 9
LD W_RANGE9_PLC2  ; ARM IN RANGE 9
AND M_Arm_Omlaag  ; Merker Arm Omlaag Plc 1 & Plc 2
OUT MRANGE9  ; IN RANGE 9
AND MRANGE9  ; IN RANGE 9
MOV(021) +1100 D_PLC2_SNELH_ARM  ; SNELHEID ARM PLC 2
MOV(021) +45 RAMP_FACTOR  ; RAMP FACTOR FOR ARM MOTION
; rung 27: copy data tbv range 10
LD W_RANGE10_PLC2  ; ARM IN RANGE 10
AND M_Arm_Omlaag  ; Merker Arm Omlaag Plc 1 & Plc 2
OUT MRANGE10  ; IN RANGE 10
AND MRANGE10  ; IN RANGE 10
MOV(021) +1500 D_PLC2_SNELH_ARM  ; SNELHEID ARM PLC 2
MOV(021) +65 RAMP_FACTOR  ; RAMP FACTOR FOR ARM MOTION

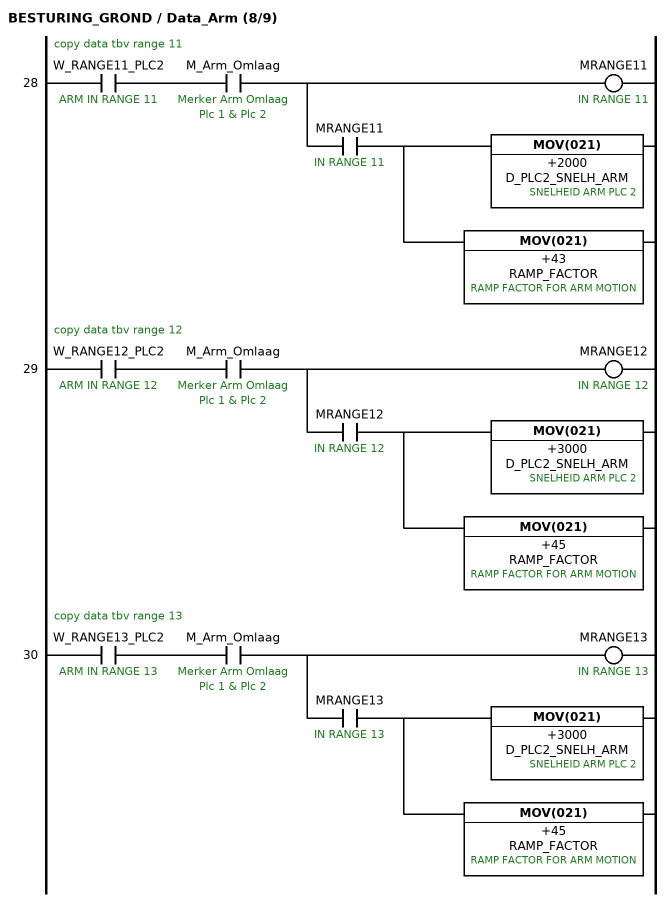
; rung 28: copy data tbv range 11
LD W_RANGE11_PLC2  ; ARM IN RANGE 11
AND M_Arm_Omlaag  ; Merker Arm Omlaag Plc 1 & Plc 2
OUT MRANGE11  ; IN RANGE 11
AND MRANGE11  ; IN RANGE 11
MOV(021) +2000 D_PLC2_SNELH_ARM  ; SNELHEID ARM PLC 2
MOV(021) +43 RAMP_FACTOR  ; RAMP FACTOR FOR ARM MOTION
; rung 29: copy data tbv range 12
LD W_RANGE12_PLC2  ; ARM IN RANGE 12
AND M_Arm_Omlaag  ; Merker Arm Omlaag Plc 1 & Plc 2
OUT MRANGE12  ; IN RANGE 12
AND MRANGE12  ; IN RANGE 12
MOV(021) +3000 D_PLC2_SNELH_ARM  ; SNELHEID ARM PLC 2
MOV(021) +45 RAMP_FACTOR  ; RAMP FACTOR FOR ARM MOTION
; rung 30: copy data tbv range 13
LD W_RANGE13_PLC2  ; ARM IN RANGE 13
AND M_Arm_Omlaag  ; Merker Arm Omlaag Plc 1 & Plc 2
OUT MRANGE13  ; IN RANGE 13
AND MRANGE13  ; IN RANGE 13
MOV(021) +3000 D_PLC2_SNELH_ARM  ; SNELHEID ARM PLC 2
MOV(021) +45 RAMP_FACTOR  ; RAMP FACTOR FOR ARM MOTION

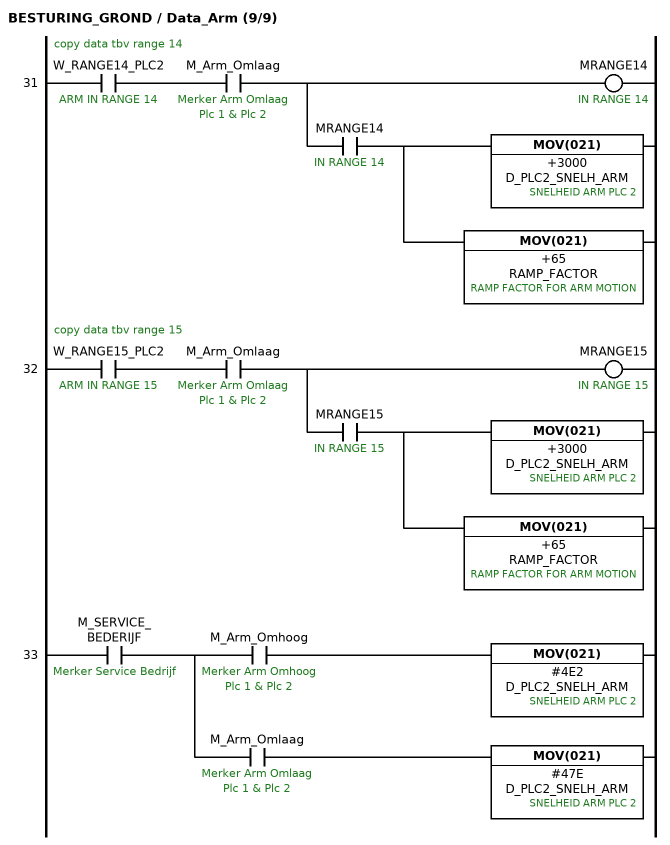
; rung 31: copy data tbv range 14
LD W_RANGE14_PLC2  ; ARM IN RANGE 14
AND M_Arm_Omlaag  ; Merker Arm Omlaag Plc 1 & Plc 2
OUT MRANGE14  ; IN RANGE 14
AND MRANGE14  ; IN RANGE 14
MOV(021) +3000 D_PLC2_SNELH_ARM  ; SNELHEID ARM PLC 2
MOV(021) +65 RAMP_FACTOR  ; RAMP FACTOR FOR ARM MOTION
; rung 32: copy data tbv range 15
LD W_RANGE15_PLC2  ; ARM IN RANGE 15
AND M_Arm_Omlaag  ; Merker Arm Omlaag Plc 1 & Plc 2
OUT MRANGE15  ; IN RANGE 15
AND MRANGE15  ; IN RANGE 15
MOV(021) +3000 D_PLC2_SNELH_ARM  ; SNELHEID ARM PLC 2
MOV(021) +65 RAMP_FACTOR  ; RAMP FACTOR FOR ARM MOTION
; rung 33
LD M_SERVICE_BEDERIJF  ; Merker Service Bedrijf
OUT TR0
AND M_Arm_Omhoog  ; Merker Arm Omhoog Plc 1 & Plc 2
MOV(021) #4E2 D_PLC2_SNELH_ARM  ; SNELHEID ARM PLC 2
LD TR0
AND M_Arm_Omlaag  ; Merker Arm Omlaag Plc 1 & Plc 2
MOV(021) #47E D_PLC2_SNELH_ARM  ; SNELHEID ARM PLC 2

### Section Besturing_Arm

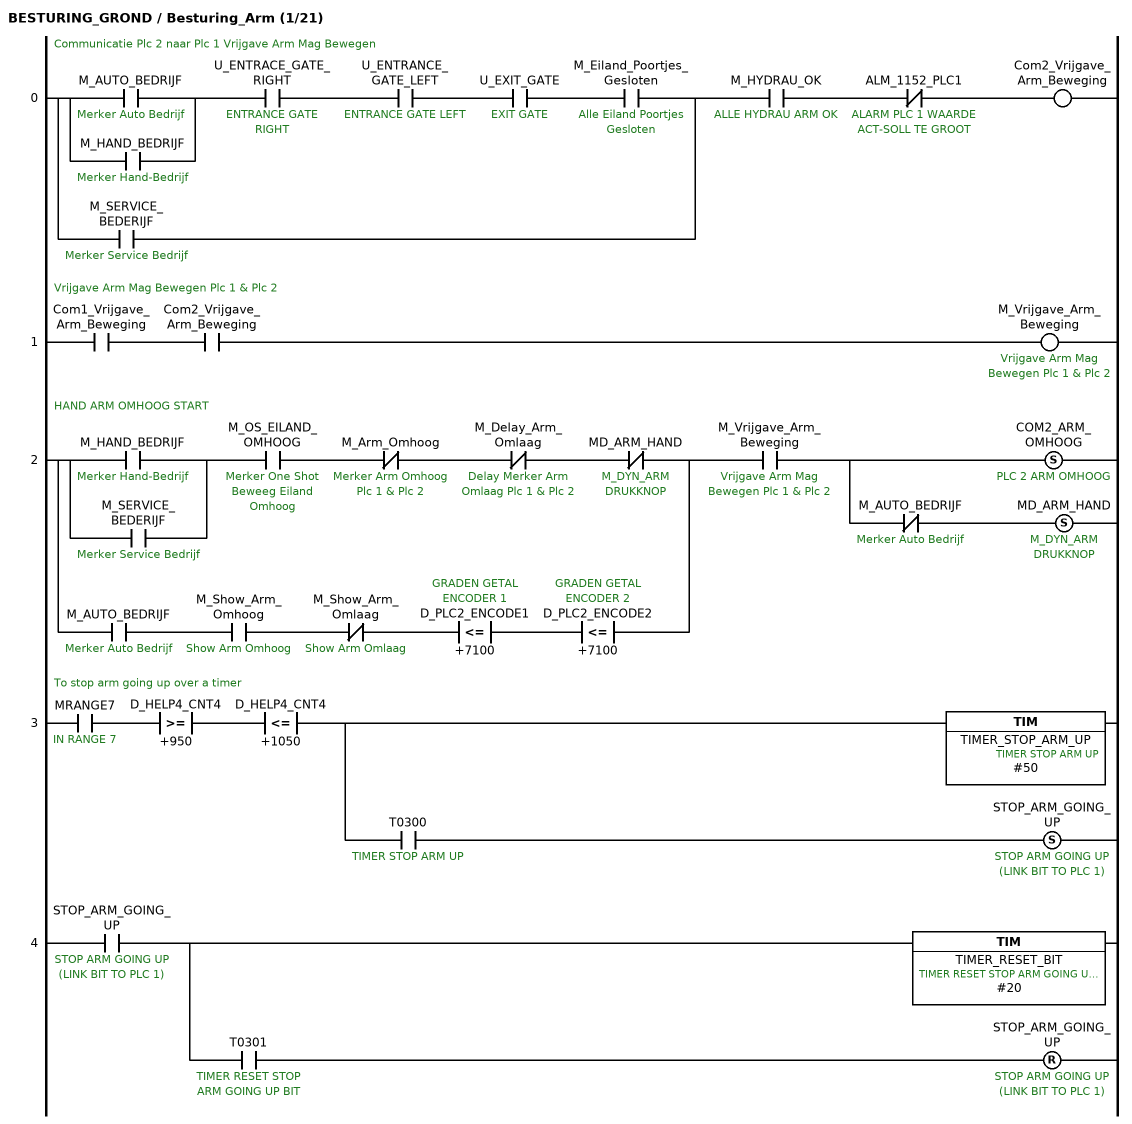
; rung 0: Communicatie Plc 2 naar Plc 1 Vrijgave Arm Mag Bewegen
LD M_AUTO_BEDRIJF  ; Merker Auto Bedrijf
OR M_HAND_BEDRIJF  ; Merker Hand-Bedrijf
AND U_ENTRACE_GATE_RIGHT  ; ENTRANCE GATE RIGHT
AND U_ENTRANCE_GATE_LEFT  ; ENTRANCE GATE LEFT
AND U_EXIT_GATE  ; EXIT GATE
AND M_Eiland_Poortjes_Gesloten  ; Alle Eiland Poortjes Gesloten
OR M_SERVICE_BEDERIJF  ; Merker Service Bedrijf
AND M_HYDRAU_OK  ; ALLE HYDRAU ARM OK
ANDNOT ALM_1152_PLC1  ; ALARM PLC 1 WAARDE ACT-SOLL TE GROOT
OUT Com2_Vrijgave_Arm_Beweging
; rung 1: Vrijgave Arm Mag Bewegen Plc 1 & Plc 2
LD Com1_Vrijgave_Arm_Beweging
AND Com2_Vrijgave_Arm_Beweging
OUT M_Vrijgave_Arm_Beweging  ; Vrijgave Arm Mag Bewegen Plc 1 & Plc 2
; rung 2: HAND ARM OMHOOG START
LD M_HAND_BEDRIJF  ; Merker Hand-Bedrijf
OR M_SERVICE_BEDERIJF  ; Merker Service Bedrijf
AND M_OS_EILAND_OMHOOG  ; Merker One Shot Beweeg Eiland Omhoog
ANDNOT M_Arm_Omhoog  ; Merker Arm Omhoog Plc 1 & Plc 2
ANDNOT M_Delay_Arm_Omlaag  ; Delay Merker Arm Omlaag Plc 1 & Plc 2
ANDNOT MD_ARM_HAND  ; M_DYN_ARM DRUKKNOP
LD M_AUTO_BEDRIJF  ; Merker Auto Bedrijf
AND M_Show_Arm_Omhoog  ; Show Arm Omhoog
ANDNOT M_Show_Arm_Omlaag  ; Show Arm Omlaag
AND<=S(317) D_PLC2_ENCODE1 +7100  ; GRADEN GETAL ENCODER 1
AND<=S(317) D_PLC2_ENCODE2 +7100  ; GRADEN GETAL ENCODER 2
ORLD
AND M_Vrijgave_Arm_Beweging  ; Vrijgave Arm Mag Bewegen Plc 1 & Plc 2
SET COM2_ARM_OMHOOG  ; PLC 2 ARM OMHOOG
ANDNOT M_AUTO_BEDRIJF  ; Merker Auto Bedrijf
SET MD_ARM_HAND  ; M_DYN_ARM DRUKKNOP
; rung 3: To stop arm going up over a timer
LD MRANGE7  ; IN RANGE 7
AND>=S(327) D_HELP4_CNT4 +950
AND<=S(317) D_HELP4_CNT4 +1050
TIM TIMER_STOP_ARM_UP #50  ; TIMER STOP ARM UP
AND T0300  ; TIMER STOP ARM UP
SET STOP_ARM_GOING_UP  ; STOP ARM GOING UP (LINK BIT TO PLC 1)
; rung 4
LD STOP_ARM_GOING_UP  ; STOP ARM GOING UP (LINK BIT TO PLC 1)
TIM TIMER_RESET_BIT #20  ; TIMER RESET STOP ARM GOING UP BIT
AND T0301  ; TIMER RESET STOP ARM GOING UP BIT
RSET STOP_ARM_GOING_UP  ; STOP ARM GOING UP (LINK BIT TO PLC 1)

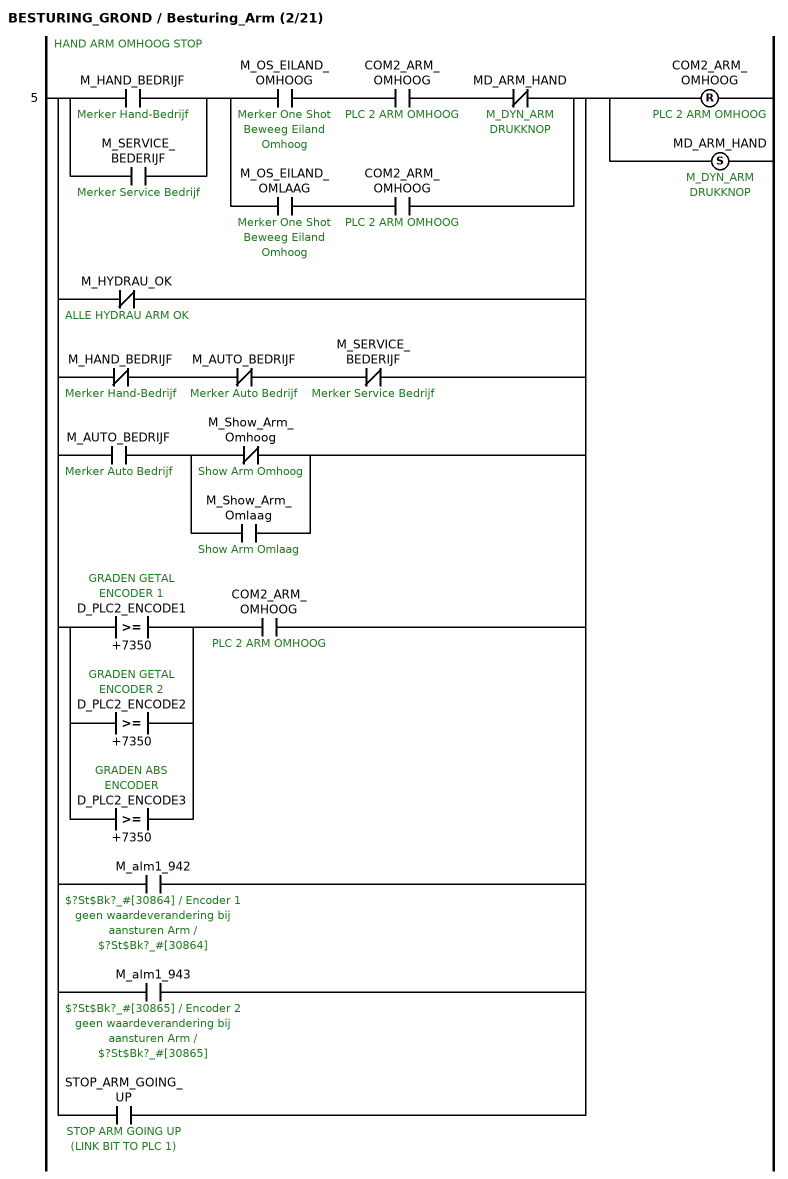
; rung 5: HAND ARM OMHOOG STOP
LD M_HAND_BEDRIJF  ; Merker Hand-Bedrijf
OR M_SERVICE_BEDERIJF  ; Merker Service Bedrijf
LD M_OS_EILAND_OMHOOG  ; Merker One Shot Beweeg Eiland Omhoog
AND COM2_ARM_OMHOOG  ; PLC 2 ARM OMHOOG
ANDNOT MD_ARM_HAND  ; M_DYN_ARM DRUKKNOP
LD M_OS_EILAND_OMLAAG  ; Merker One Shot Beweeg Eiland Omhoog
AND COM2_ARM_OMHOOG  ; PLC 2 ARM OMHOOG
ORLD
ANDLD
ORNOT M_HYDRAU_OK  ; ALLE HYDRAU ARM OK
LDNOT M_HAND_BEDRIJF  ; Merker Hand-Bedrijf
ANDNOT M_AUTO_BEDRIJF  ; Merker Auto Bedrijf
ANDNOT M_SERVICE_BEDERIJF  ; Merker Service Bedrijf
ORLD
LD M_AUTO_BEDRIJF  ; Merker Auto Bedrijf
LDNOT M_Show_Arm_Omhoog  ; Show Arm Omhoog
OR M_Show_Arm_Omlaag  ; Show Arm Omlaag
ANDLD
ORLD
LD>=S(327) D_PLC2_ENCODE1 +7350  ; GRADEN GETAL ENCODER 1
OR>=S(327) D_PLC2_ENCODE2 +7350  ; GRADEN GETAL ENCODER 2
OR>=S(327) D_PLC2_ENCODE3 +7350  ; GRADEN ABS ENCODER
AND COM2_ARM_OMHOOG  ; PLC 2 ARM OMHOOG
ORLD
OR M_alm1_942  ; $?St$Bk?_#[30864] / Encoder 1 geen waardeverandering bij aansturen Arm / $?St$Bk?_#[30864]
OR M_alm1_943  ; $?St$Bk?_#[30865] / Encoder 2 geen waardeverandering bij aansturen Arm / $?St$Bk?_#[30865]
OR STOP_ARM_GOING_UP  ; STOP ARM GOING UP (LINK BIT TO PLC 1)
RSET COM2_ARM_OMHOOG  ; PLC 2 ARM OMHOOG
SET MD_ARM_HAND  ; M_DYN_ARM DRUKKNOP

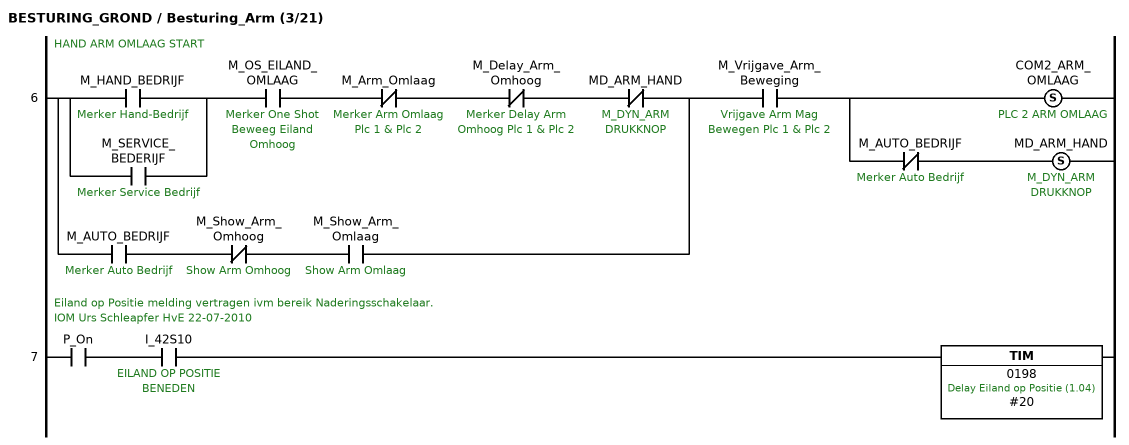
; rung 6: HAND ARM OMLAAG START
LD M_HAND_BEDRIJF  ; Merker Hand-Bedrijf
OR M_SERVICE_BEDERIJF  ; Merker Service Bedrijf
AND M_OS_EILAND_OMLAAG  ; Merker One Shot Beweeg Eiland Omhoog
ANDNOT M_Arm_Omlaag  ; Merker Arm Omlaag Plc 1 & Plc 2
ANDNOT M_Delay_Arm_Omhoog  ; Merker Delay Arm Omhoog Plc 1 & Plc 2
ANDNOT MD_ARM_HAND  ; M_DYN_ARM DRUKKNOP
LD M_AUTO_BEDRIJF  ; Merker Auto Bedrijf
ANDNOT M_Show_Arm_Omhoog  ; Show Arm Omhoog
AND M_Show_Arm_Omlaag  ; Show Arm Omlaag
ORLD
AND M_Vrijgave_Arm_Beweging  ; Vrijgave Arm Mag Bewegen Plc 1 & Plc 2
SET COM2_ARM_OMLAAG  ; PLC 2 ARM OMLAAG
ANDNOT M_AUTO_BEDRIJF  ; Merker Auto Bedrijf
SET MD_ARM_HAND  ; M_DYN_ARM DRUKKNOP
; rung 7: Eiland op Positie melding vertragen ivm bereik Naderingsschakelaar. / IOM Urs Schleapfer HvE 22-07-2010
LD P_On
AND I_42S10  ; EILAND OP POSITIE BENEDEN
TIM 0198 #20  ; Delay Eiland op Positie (1.04)

